W155.13 BOOL  ; EMERG STOP:DEVICE NET COMMUNICATION ABNORMALITY
W155.14 BOOL  ; Servo Carrier Transfer Error
W156.00 BOOL  ; AUTO STOP:INSULATION TESTER FAULT
W156.01 BOOL  ; AUTO STOP:RESISTANCE TESTER FAULT
W156.02 BOOL  ; AUTO STOP:IMPULSE TESTER FAULT
W158.00 BOOL  ; CYCLE STOP:QUALITY CHECK
W159.01 BOOL  ; CYCLE STOP:CONTACT PROBE IN WITHSTAND VOLTAGE FAULT
W159.02 BOOL  ; CYCLE STOP:INSULATION TEST FAULT CONTINUALING
W159.03 BOOL  ; CYCLE STOP:WORK No. FAULT CONTINUALING
W159.04 BOOL  ; CYCLE STOP:SWING MEASUREMENT FAULT CONTINUALING
W159.05 BOOL  ; CYCLE STOP:RESISTANCE MEASUREMENT FAULT CONTINUALING
W159.06 BOOL  ; CYCLE STOP:PAIR POLE IMPULSE MEAS FAULT CONTINUALING
W159.07 BOOL  ; CYCLE STOP:NEXT POLE IMPULSE MEAS FAULT CONTINUALING
W159.08 BOOL  ; CYCLE STOP:LENGTH MEASUREMENT FAULT CONTINUALING
W159.09 BOOL  ; CYCLE STOP:THICKNESS OF CORE FAULT CONTINUALING
W159.10 BOOL  ; CYCLE STOP:COIL END FAULT CONTINUALING
W159.11 BOOL  ; CYCLE STOP:WITHSTAND VOLTAGE CONTACT PROBE CHANGE
W159.12 BOOL  ; CYCLE STOP:RESISTANCE CONTACT PROBE CHANGE
W159.13 BOOL  ; CYCLE STOP:IMPULSE CONTACT PROBE CHANGE
W159.14 BOOL  ; CYCLE STOP:BEARING INSIDE AND OUTSIDE CHECK NG
W159.15 BOOL  ; CYCLE STOP:FULL FRACTION TRAY
W160.00 BOOL  ; CYCLE STOP:LOADING WORKPIECE CLAMP FAULT
W160.01 BOOL  ; CYCLE STOP:UNLOADING WORKPIECE CLAMP FAULT
W160.02 BOOL  ; CYCLE STOP:BEARING MEASUREMENT FAULT CONTINUALING
W160.03 BOOL  ; -
W161.00 BOOL  ; CYCLE STOP:NO WORK No. SWITCH NEXT PRODUCT WORK No.
W163.01 BOOL  ; FAULT STOP:LOADING C/V CYCLE TIME OVER
W163.02 BOOL  ; FAULT STOP:LOADER CYCLE TIME OVER
W163.03 BOOL  ; FAULT STOP:TRANSFER CARRIER CYCLE TIME OVER
W163.04 BOOL  ; FAULT STOP:FWORKPIECE PUSHER CYCLE TIME OVER
W163.05 BOOL  ; FAULT STOP:INSULATION TEST CYCLE TIME OVER
W163.06 BOOL  ; FAULT STOP:SWING MEASUREMENT CYCLE TIME OVER
W163.07 BOOL  ; FAULT STOP:RESISTANCE CYCLE TIME OVER
W163.08 BOOL  ; FAULT STOP:IMPULSE CYCLE TIME OVER
W163.09 BOOL  ; FAULT STOP:BEARING INSERT CYCLE TIME OVER
W163.10 BOOL  ; FAULT STOP:LENGTH MEASUREMENT CYCLE TIME OVER
W163.11 BOOL  ; FAULT STOP:UNLOADING CYCLE TIME OVER
W163.12 BOOL  ; FAULT STOP:BEARING SUPPLY CYCLE TIME OVER
W163.13 BOOL  ; FAULT STOP:BEARING EXCHANGE CYCLE TIME OVER
W163.14 BOOL  ; FAULT STOP:DEFECT DISCHARGE CYCLE TIME OVER
W163.15 BOOL  ; FAULT STOP:LANE 1 PALLETIZING CYCLE TIME OVER
W164.00 BOOL  ; FAULT STOP:LANE 1 SUPPLYING CYCLE TIME OVER
W164.01 BOOL  ; FAULT STOP:LANE 1 STACKING CYCLE TIME OVER
W164.02 BOOL  ; FAULT STOP:LANE 2 PALLETIZING CYCLE TIME OVER
W164.03 BOOL  ; FAULT STOP:LANE 2 SUPPLYING CYCLE TIME OVER
W164.04 BOOL  ; FAULT STOP:LANE 2 STACKING CYCLE TIME OVER
W164.07 BOOL  ; -
W164.08 BOOL  ; -
W166.00 BOOL  ; PAUSE:FULL WORKPIECES OF DEFECT DISCHARGING C/V
W166.01 BOOL  ; PAUSE:LANE 1 FULL UNLOADING CONTAINER
W166.02 BOOL  ; PAUSE:LANE 2 FULL UNLOADING CONTAINER
W166.04 BOOL  ; PAUSE:LANE 1 FULL BEARING TRAY
W166.05 BOOL  ; PAUSE:LANE 1 SHORTAGE OF LOADING CONTAINER
W166.06 BOOL  ; PAUSE:LANE 2 SHORTAGE OF LOADING CONTAINER
W166.08 BOOL  ; PAUSE:SHORTAGE OF BEARING TRAY
W167.00 BOOL  ; NOTICE OF STOP:QUALITY CHECK
W167.01 BOOL  ; NOTICE OF STOP:WITHSTAND VOLTAGE CONTACT PROBE CHANGE
W167.02 BOOL  ; NOTICE OF STOP:RESISTANCE CONTACT PROBE CHANGE
W167.03 BOOL  ; NOTICE OF STOP:IMPULSE CONTACT PROBE CHANGE
W168.00 BOOL  ; PAUSE:WAITING FOR LOADING WORKPIECE
W169.00 BOOL  ; WARNING:SAFETY GUARD OPEN
W169.01 BOOL  ; WARNING:ID COLLATION FAULT OF LOADING CONTAINER
W169.02 BOOL  ; WARNING:SWITCH NEXT WORK No. UNSETTING
W169.03 BOOL  ; WARNING:NO RESPONSE OF ID1
W169.04 BOOL  ; WARNING:COMMUNICATION FAULT OF ID 1
W169.05 BOOL  ; WARNING:NO RESPONSE OF ID2
W169.06 BOOL  ; WARNING:COMMUNICATION FAULT OF ID 2
W169.07 BOOL  ; WARNING:NO RESPONSE OF ID3
W169.08 BOOL  ; WARNING:COMMUNICATION FAULT OF ID 3
W169.09 BOOL  ; WARNING:NO RESPONSE OF ID4
W169.10 BOOL  ; WARNING:COMMUNICATION FAULT OF ID 4
W169.13 BOOL  ; WARNING:BEARING ROBOT BAATERY CHANGE
W169.14 BOOL  ; WARNING:UNLOADING ROBOT BAATERY CHANGE
W169.15 BOOL  ; WARNING:PC BAATERY CHANGE
W170.00 BOOL  ; Defective history clearness
W171.00 BOOL  ; DATA CLEAR
W172.00 BOOL  ; DATA CLEAR
W173.00 BOOL  ; Fraction palette data clearness
W173.11 BOOL  ; Counter effective PB of time
W173.12 BOOL  ; Counter invalid PB of time
W173.13 BOOL  ; Data reset
W173.14 BOOL  ; Stop at one o'clock of utilization rates meter
W174.00 BOOL  ; WORKPIECE MEMORY CLEAR (CORE DISTINCTION UNIT)
W174.01 BOOL  ; WORKPIECE MEMORY CLEAR (INSULATION UNIT)
W174.02 BOOL  ; WORKPIECE MEMORY CLEAR (SWING MEASUREMENT UNIT)
W174.03 BOOL  ; WORKPIECE MEMORY CLEAR (RESISTANCE MEASUREMENT UNIT)
W174.04 BOOL  ; WORKPIECE MEMORY CLEAR (IMPULSE MEASUREMENT UNIT)
W174.05 BOOL  ; WORKPIECE MEMORY CLEAR (BEARING INSERT UNIT)
W174.06 BOOL  ; WORKPIECE MEMORY CLEAR (LENGTH MEASUREMENT UNIT)
W174.07 BOOL  ; WORKPIECE MEMORY CLEAR (UNLOADING UNIT)
W174.08 BOOL  ; WORKPIECE MEMORY CLEAR (ROBOT CHUCK)
W175.10 BOOL  ; Stop at one o'clock of utilization rates meter
W175.11 BOOL  ; Counter effective inside of time
W175.12 BOOL  ; Counter invalid inside of time
W175.14 BOOL  ; It is stopping at one o'clock of the utilization rates meter.
W176.00 BOOL  ; SHORT STOP DATA CLEAR
W176.01 BOOL  ; NO STOP TIME CLEAR
W176.02 BOOL  ; ARMATURE LINE RUNNING
W176.03 BOOL  ; NO STOP TIME COUNT
W176.05 BOOL  ; -
W176.06 BOOL  ; -
W176.07 BOOL  ; -
W176.08 BOOL  ; -
W176.09 BOOL  ; -
W176.10 BOOL  ; -
W18.00 BOOL  ; 11ST_HOME POSITION RETURN PUSH BUTTON SWITCH
W18.01 BOOL  ; 12ST_HOME POSITION RETURN PUSH BUTTON SWITCH
W18.02 BOOL  ; 13ST_HOME POSITION RETURN PUSH BUTTON SWITCH
W18.03 BOOL  ; 14ST_HOME POSITION RETURN PUSH BUTTON SWITCH
W18.04 BOOL  ; 15ST_HOME POSITION RETURN PUSH BUTTON SWITCH
W18.05 BOOL  ; 16ST_HOME POSITION RETURN PUSH BUTTON SWITCH
W18.06 BOOL  ; 17ST_HOME POSITION RETURN PUSH BUTTON SWITCH
W18.07 BOOL  ; 18ST_HOME POSITION RETURN PUSH BUTTON SWITCH
W18.08 BOOL  ; 19ST_HOME POSITION RETURN PUSH BUTTON SWITCH
W18.09 BOOL  ; 20ST_HOME POSITION RETURN PUSH BUTTON SWITCH
W190.00 BOOL  ; ALARM (1ST) PL
W190.01 BOOL  ; ALARM (2ST) PL
W190.02 BOOL  ; ALARM (3ST) PL
W190.03 BOOL  ; ALARM (4ST) PL
W190.04 BOOL  ; ALARM (5ST) PL
W190.05 BOOL  ; ALARM (6ST) PL
W190.06 BOOL  ; ALARM (7ST) PL
W190.07 BOOL  ; ALARM (8ST) PL
W190.08 BOOL  ; ALARM (9ST) PL
W190.09 BOOL  ; ALARM (10ST) PL
W190.10 BOOL  ; ALARM (11ST) PL
W190.11 BOOL  ; ALARM (12ST) PL
W190.12 BOOL  ; ALARM (13ST) PL
W190.13 BOOL  ; ALARM (14ST) PL
W190.14 BOOL  ; ALARM (15ST) PL
W190.15 BOOL  ; ALARM (16ST) PL
W191.00 BOOL  ; CAUTION (1ST) PL
W191.01 BOOL  ; CAUTION (2ST) PL
W191.02 BOOL  ; CAUTION (3ST) PL
W191.03 BOOL  ; CAUTION (4ST) PL
W191.04 BOOL  ; CAUTION (5ST) PL
W191.05 BOOL  ; CAUTION (6ST) PL
W191.06 BOOL  ; CAUTION (7ST) PL
W191.07 BOOL  ; CAUTION (8ST) PL
W191.08 BOOL  ; CAUTION (9ST) PL
W191.09 BOOL  ; CAUTION (10ST) PL
W191.10 BOOL  ; CAUTION (11ST) PL
W191.11 BOOL  ; CAUTION (12ST) PL
W191.12 BOOL  ; CAUTION (13ST) PL
W191.13 BOOL  ; CAUTION (14ST) PL
W191.14 BOOL  ; CAUTION (15ST) PL
W191.15 BOOL  ; CAUTION (16ST) PL
W192.00 BOOL  ; NO FAULT (1ST) PL
W192.01 BOOL  ; NO FAULT (2ST) PL
W192.02 BOOL  ; NO FAULT (3ST) PL
W192.03 BOOL  ; NO FAULT (4ST) PL
W192.04 BOOL  ; NO FAULT (5ST) PL
W192.05 BOOL  ; NO FAULT (6ST) PL
W192.06 BOOL  ; NO FAULT (7ST) PL
W192.07 BOOL  ; NO FAULT (8ST) PL
W192.08 BOOL  ; NO FAULT (9ST) PL
W192.09 BOOL  ; NO FAULT (10ST) PL
W192.10 BOOL  ; NO FAULT (11ST) PL
W192.11 BOOL  ; NO FAULT (12ST) PL
W192.12 BOOL  ; NO FAULT (13ST) PL
W192.13 BOOL  ; NO FAULT (14ST) PL
W192.14 BOOL  ; NO FAULT (15ST) PL
W192.15 BOOL  ; NO FAULT (16ST) PL
W193.00 BOOL  ; ALARM (17ST) PL
W193.01 BOOL  ; ALARM (18ST) PL
W193.02 BOOL  ; ALARM (19ST) PL
W193.03 BOOL  ; ALARM (20ST) PL
W194.00 BOOL  ; CAUTION (17ST) PL
W194.01 BOOL  ; CAUTION (18ST) PL
W194.02 BOOL  ; CAUTION (19ST) PL
W194.03 BOOL  ; CAUTION (20ST) PL
W195.00 BOOL  ; NO FAULT (17ST) PL
W195.01 BOOL  ; NO FAULT (18ST) PL
W195.02 BOOL  ; NO FAULT (19ST) PL
W195.03 BOOL  ; NO FAULT (20ST) PL
W199.08 BOOL  ; SHORT STOP HISTORY SAVE
W199.09 BOOL  ; SHORT STOP HISTORY SAVING
W199.10 BOOL  ; SHORT STOP HISTORY SAVE COMPLETE
W199.11 BOOL  ; SHORT STOP HISTORY SAVE PERMIT
W199.12 BOOL  ; FAULT STOP HISTORY SAVE
W199.13 BOOL  ; FAULT STOP HISTORY SAVING
W199.14 BOOL  ; FAULT STOP HISTORY SAVE COMPLETE
W199.15 BOOL  ; FAULT STOP HISTORY SAVE PERMIT
W19.00 BOOL  ; 11ST_HOME POSITION/RUNNING
W19.01 BOOL  ; 12ST_HOME POSITION/RUNNING
W19.02 BOOL  ; 13ST_HOME POSITION/RUNNING
W19.03 BOOL  ; 14ST_HOME POSITION/RUNNING
W19.04 BOOL  ; 15ST_HOME POSITION/RUNNING
W19.05 BOOL  ; 16ST_HOME POSITION/RUNNING
W19.06 BOOL  ; 17ST_HOME POSITION/RUNNING
W19.07 BOOL  ; 18ST_HOME POSITION/RUNNING
W19.08 BOOL  ; 19ST_HOME POSITION/RUNNING
W19.09 BOOL  ; 20ST_HOME POSITION/RUNNING
W1.00 BOOL  ; MASTER SWITCH ON
W1.01 BOOL  ; AUTO RUNNING
W1.02 BOOL  ; CYCLE STOP
W1.03 BOOL  ; ALL HOME POSITION
W1.04 BOOL  ; OPERATION AUTOMATIC SELECT
W1.05 BOOL  ; OPERATION INDIVIDUAL SELECT
W1.06 BOOL  ; ROBOT 1 RUNNING
W1.07 BOOL  ; ROBOT 2 RUNNING
W1.08 BOOL  ; LS203115
W1.09 BOOL  ; Safety cover invalidity PL
W20.00 BOOL  ; 01ST_HOME POSITION RETURN PUSH BUTTON SWITCH
W20.01 BOOL  ; 02ST_HOME POSITION RETURN PUSH BUTTON SWITCH
W20.02 BOOL  ; 03ST_HOME POSITION RETURN PUSH BUTTON SWITCH
W20.03 BOOL  ; 04ST_HOME POSITION RETURN PUSH BUTTON SWITCH
W20.04 BOOL  ; 05ST_HOME POSITION RETURN PUSH BUTTON SWITCH
W20.05 BOOL  ; 06ST_HOME POSITION RETURN PUSH BUTTON SWITCH
W20.06 BOOL  ; 07ST_HOME POSITION RETURN PUSH BUTTON SWITCH
W20.07 BOOL  ; 08ST_HOME POSITION RETURN PUSH BUTTON SWITCH
W20.08 BOOL  ; 09ST_HOME POSITION RETURN PUSH BUTTON SWITCH
W20.09 BOOL  ; 10ST_HOME POSITION RETURN PUSH BUTTON SWITCH
W21.00 BOOL  ; 01ST_HOME POSITION/RUNNING
W21.01 BOOL  ; 02ST_HOME POSITION/RUNNING
W21.02 BOOL  ; 03ST_HOME POSITION/RUNNING
W21.03 BOOL  ; 04ST_HOME POSITION/RUNNING
W21.04 BOOL  ; 05ST_HOME POSITION/RUNNING
W21.05 BOOL  ; 06ST_HOME POSITION/RUNNING
W21.06 BOOL  ; 07ST_HOME POSITION/RUNNING
W21.07 BOOL  ; 08ST_HOME POSITION/RUNNING
W21.08 BOOL  ; 09ST_HOME POSITION/RUNNING
W21.09 BOOL  ; 10ST_HOME POSITION/RUNNING
W25.00 BOOL  ; LOADING CONVEYOR PALLET SHIFT FORWARD
W25.01 BOOL  ; LOADING CONVEYOR PALLET SHIFT BACKWARD
W25.04 BOOL  ; LOADING CONVEYOR PALLET DISCHARGE FORWARD
W25.05 BOOL  ; LOADING CONVEYOR PALLET DISCHARGE BACKWARD
W26.00 BOOL  ; LOADING CONVEYOR PALLET SHIFT FORWARD END
W26.01 BOOL  ; LOADING CONVEYOR PALLET SHIFT BACKWARD END
W26.04 BOOL  ; LOADING CONVEYOR PALLET DISCHARGE FORWARD END
W26.05 BOOL  ; LOADING CONVEYOR PALLET DISCHARGE BACKWARD END
W27.00 BOOL  ; WORKPIECE ON FORMER PROCESS
W27.10 BOOL  ; 01ST_1CY START PB
W27.11 BOOL  ; 01ST_1CY RUN PL
W27.12 BOOL  ; 01ST_UNIT HOME POSITION RETURN PB
W27.13 BOOL  ; 01ST_UNIT HOME POSITION PL
W28.00 BOOL  ; LOADER FORWARD
W28.01 BOOL  ; LOADER BACKWARD
W28.02 BOOL  ; LOADER DOWNWARD
W28.03 BOOL  ; LOADER UPWARD
W28.04 BOOL  ; TURN LOADER CHUCK TURN
W28.05 BOOL  ; TURN LOADER RECHUCK TURN
W28.06 BOOL  ; LOADER CHUCK CLAMP
W28.07 BOOL  ; LOADER CHUCK UNCLAMP
W29.00 BOOL  ; LOADER FORWARD END
W29.01 BOOL  ; LOADER BACKWARD END
W29.02 BOOL  ; LOADER DOWNWARD END
W29.03 BOOL  ; LOADER UPWARD END
W29.04 BOOL  ; TURN LOADER CHUCK TURN END
W29.05 BOOL  ; TURN LOADER CHUCK RETURN END
W29.06 BOOL  ; LOADER CHUCK CLAMP END
W29.07 BOOL  ; LOADER CHUCK UNCLAMP END
W2.01 BOOL  ; $?St$Bk?_#[22] / PB_Upper limit master check / $?St$Bk?_#[22]
W2.02 BOOL  ; ROBOT MASTER ON
W2.03 BOOL  ; ROBOT FIXED POSITION RETURN
W2.04 BOOL  ; LENGTH MASTER O SETTING
W2.05 BOOL  ; BEARING FIXID POSITION RETURN
W2.06 BOOL  ; ALL MACHINES SAVING ENERGY OF FLURESCENT LIGHT
W2.07 BOOL  ; PB_Lower limit master check
W2.09 BOOL  ; LANGUAGE CHANGE PB
W2.10 BOOL  ; SAVING ENERGY OF FLURESCENT LIGHT
W300.00 BOOL  ; Piling up one lane step lot end(four steps)
W300.01 BOOL  ; Piling up two lane step lot end(four steps)
W300.02 BOOL  ; ID RESET START SELECT PB ON
W300.03 BOOL  ; ID RESET START
W300.04 BOOL  ; ID RESET RUNNING
W301.00 BOOL  ; TEMPORARY CONTACT FOR ADJUSTMENT ON
W301.01 BOOL  ; Product number change 1 （for disp）
W301.02 BOOL  ; Crear product number change 1 （for disp）
W301.05 BOOL  ; -
W301.06 BOOL  ; -
W301.10 BOOL  ; -
W301.15 BOOL  ; 調整用仮接点（ﾜｰｸ押さえ上昇ﾀｲﾐﾝｸﾞ）
W302.01 BOOL  ; Product number change 2 （for disp）
W302.02 BOOL  ; Crear product number change 2 （for disp）
W302.10 BOOL  ; -
W30.00 BOOL  ; TRANSFER CARRIER NO INTERFERENCE
W30.10 BOOL  ; 02ST_1CY START PB
W30.11 BOOL  ; 02ST_1CY RUN PL
W30.12 BOOL  ; 02ST_UNIT HOME POSITION RETURN PB
W30.13 BOOL  ; 02ST_UNIT HOME POSITION PL
W31.00 BOOL  ; TRANSFER CARRIER LIFT UPWARD
W31.01 BOOL  ; TRANSFER CARRIER LIFT DOWNWARD
W31.02 BOOL  ; TRANSFER CARRIER FORWARD
W31.03 BOOL  ; TRANSFER CARRIER BACKWARD
W32.00 BOOL  ; TRANSFER CARRIER LIFT UPWARD END
W32.01 BOOL  ; TRANSFER CARRIER LIFT DOWNWARD END
W32.02 BOOL  ; TRANSFER CARRIER FORWARD END
W32.03 BOOL  ; TRANSFER CARRIER BACKWARD END
W33.00 BOOL  ; Completion of distinction of thickness in core
W33.01 BOOL  ; INSULATION TEST COMPLETE
W33.02 BOOL  ; SWING & COIL END COMPLETE
W33.03 BOOL  ; RESISTANCE MEASUREMENT COMPLETE
W33.04 BOOL  ; IMPULSE COMPLETE
W33.05 BOOL  ; BEARING INSERT COMPLETE
W33.06 BOOL  ; LENGTH CHECK COMPLETE
W33.10 BOOL  ; 03ST_1CY START PB
W33.11 BOOL  ; 03ST_1CY RUN PL
W33.12 BOOL  ; 03ST_UNIT HOME POSITION RETURN PB
W33.13 BOOL  ; 03ST_UNIT HOME POSITION PL
W34.00 BOOL  ; WORKPIECE PUSHER FORWARD
W34.01 BOOL  ; WORKPIECE PUSHER BACKWARD
W34.04 BOOL  ; Start of distinction of thickness in core
W34.05 BOOL  ; Stop of distinction of thickness in core
W350.00 BOOL  ; -
W351.00 BOOL  ; -
W35.00 BOOL  ; WORKPIECE PUSHER FORWARD
W35.01 BOOL  ; WORKPIECE PUSHER BACKWARD
W35.04 BOOL  ; Start of distinction of thickness in core
W35.05 BOOL  ; Stop of distinction of thickness in core
W36.01 BOOL  ; Completion of distinction of thickness in core
W36.10 BOOL  ; 04ST_1CY START PB
W36.11 BOOL  ; 04ST_1CY RUN PL
W36.12 BOOL  ; 04ST_UNIT HOME POSITION RETURN PB
W36.13 BOOL  ; 04ST_UNIT HOME POSITION PL
W37.00 BOOL  ; TRANSFER CARRIER LIFT UPWARD
W37.01 BOOL  ; TRANSFER CARRIER LIFT DOWNWARD
W37.04 BOOL  ; INSULATION TEST START
W37.05 BOOL  ; INSULATION TEST STOP
W38.00 BOOL  ; TRANSFER CARRIER LIFT UPWARD END
W38.01 BOOL  ; TRANSFER CARRIER LIFT DOWNWARD END
W38.04 BOOL  ; INSULATION TEST START
W38.05 BOOL  ; INSULATION TEST STOP
W39.01 BOOL  ; INSULATION TEST OK
W39.02 BOOL  ; INSULATION TEST NG
W39.03 BOOL  ; INSULATION TEST COMPLETE
W39.10 BOOL  ; 05ST_1CY START PB
W39.11 BOOL  ; 05ST_1CY RUN PL
W39.12 BOOL  ; 05ST_UNIT HOME POSITION RETURN PB
W39.13 BOOL  ; 05ST_UNIT HOME POSITION PL
W3.01 BOOL  ; PL_Upper limit check completed (functional check)
W3.02 BOOL  ; ROBOT MASTER ON
W3.03 BOOL  ; ROBOT FIXED POSITION PL
W3.04 BOOL  ; PL_LENGTH 0 MASTER SETTING
W3.05 BOOL  ; BEARING FIXID POSITION PL
W3.06 BOOL  ; ALL MACHINES SAVING ENERGY OF FLURESCENT LIGHT
W3.07 BOOL  ; PL_Lower limit check completed (functional check)
W3.10 BOOL  ; SAVING ENERGY OF FLURESCENT LIGHT
W3.11 BOOL  ; SAVING ENERGY OF FLURESCENT LIGHT
W400.00 BOOL  ; TRANSFER +JOG
W400.01 BOOL  ; TRANSFER -JOG
W400.03 BOOL  ; FORWARD POSITION S
W400.04 BOOL  ; BACKWARD POSITION S
W400.07 BOOL  ; Set Up
W400.15 BOOL  ; POSITIONAL DATA CAN BE INPUT
W40.00 BOOL  ; TRANSFER CARRIER LIFT UPWARD
W40.01 BOOL  ; TRANSFER CARRIER LIFT DOWNWARD
W40.02 BOOL  ; POSITIONING ARROW FORWARD
W40.03 BOOL  ; POSITIONING ARROW BACKWARD
W40.04 BOOL  ; POSITIONING START
W40.05 BOOL  ; POSITIONING STOP
W40.08 BOOL  ; SWING MEASURE START
W40.09 BOOL  ; SWING MEASURE STOP
W41.00 BOOL  ; TRANSFER CARRIER LIFT UPWARD END
W41.01 BOOL  ; TRANSFER CARRIER LIFT DOWNWARDD END
W41.02 BOOL  ; POSITIONING ARROW FORWARDD END
W41.03 BOOL  ; POSITIONING ARROW BACKWARDD END
W41.04 BOOL  ; POSITIONING START
W41.05 BOOL  ; POSITIONING STOP
W41.08 BOOL  ; SWING MEASURE START
W41.09 BOOL  ; SWING MEASURE STOP
W42.01 BOOL  ; SWING OK
W42.02 BOOL  ; SWING NG
W42.03 BOOL  ; SWING & COIL END COMPLETE
W42.10 BOOL  ; 06ST_1CY START PB
W42.11 BOOL  ; 06ST_1CY RUN PL
W42.12 BOOL  ; 06ST_UNIT HOME POSITION RETURN PB
W42.13 BOOL  ; 06ST_UNIT HOME POSITION PL
W43.02 BOOL  ; WORKPIECE CLAMP DOWNWARD
W43.03 BOOL  ; WORKPIECE CLAMP UPWARD
W43.06 BOOL  ; TRANSFER CARRIER LIFT UPWARD
W43.07 BOOL  ; TRANSFER CARRIER LIFT DOWNWARD
W43.10 BOOL  ; CONTACT PROBE IN RESISTANCE FORWARD
W43.11 BOOL  ; CONTACT PROBE IN RESISTANCE BACKWARD
W43.14 BOOL  ; RESISTANCE MEASUREMENT START
W43.15 BOOL  ; RESISTANCE MEASUREMENT STOP
W44.02 BOOL  ; TRANSFER CARRIER LIFT UPWARD END
W44.03 BOOL  ; TRANSFER CARRIER LIFT DOWNWARD END
W44.06 BOOL  ; CONTACT PROBE IN RESISTANCE FORWARD END
W44.07 BOOL  ; CONTACT PROBE IN RESISTANCE BACKWARD END
W44.10 BOOL  ; CONTACT PROBE IN RESISTANCE FORWARD END
W44.11 BOOL  ; CONTACT PROBE IN RESISTANCE BACKWARD END
W44.14 BOOL  ; RESISTANCE MEASUREMENT START
W44.15 BOOL  ; RESISTANCE MEASUREMENT STOP
W45.01 BOOL  ; RESISTANCE OK (80)
W45.02 BOOL  ; RESISTANCE NG (80)
W45.03 BOOL  ; RESISTANCE OK (180)
W45.04 BOOL  ; RESISTANCE NG (180)
W45.05 BOOL  ; RESISTANCE MEASUREMENT COMPLETE
W45.10 BOOL  ; 07ST_1CY START PB
W45.11 BOOL  ; 07ST_1CY RUN PL
W45.12 BOOL  ; 07ST_UNIT HOME POSITION RETURN PB
W45.13 BOOL  ; 07ST_UNIT HOME POSITION PL
W46.00 BOOL  ; WORKPIECE CLAMP DOWNWARD
W46.01 BOOL  ; WORKPIECE CLAMP UPWARD
W46.02 BOOL  ; CONTACT PROBE IN INPULSE FORWARD
W46.03 BOOL  ; CONTACT PROBE IN INPULSE BACKWARD
W46.04 BOOL  ; TRANSFER CARRIER LIFT UPWARD
W46.05 BOOL  ; TRANSFER CARRIER LIFT DOWNWARD
W46.06 BOOL  ; IMPULSE MEASUREMENT START
W46.07 BOOL  ; IMPULSE MEASUREMENT STOP
W46.09 BOOL  ; WABE INDICATION
W46.10 BOOL  ; Relay ON to pair pole
W46.11 BOOL  ; Relay ON to next pole
W46.14 BOOL  ; STEP MODE ON
W46.15 BOOL  ; STEP UP
W47.00 BOOL  ; WORKPIECE CLAMP DOWNWARD END
W47.01 BOOL  ; WORKPIECE CLAMP UPWARD END
W47.02 BOOL  ; CONTACT PROBE IN INPULSE FORWARD END
W47.03 BOOL  ; CONTACT PROBE IN INPULSE BACKWARD END
W47.04 BOOL  ; TRANSFER CARRIER LIFT UPWARD END
W47.05 BOOL  ; TRANSFER CARRIER LIFT DOWNWARD END
W47.06 BOOL  ; IMPULSE MEASUREMENT START
W47.07 BOOL  ; IMPULSE MEASUREMENT STOP
W47.09 BOOL  ; WABE INDICATION
W47.10 BOOL  ; Relay ON to pair pole
W47.11 BOOL  ; Relay ON to next pole
W47.14 BOOL  ; STEP MODE ON
W47.15 BOOL  ; STEP UP
W48.01 BOOL  ; PAIR POLE OK
W48.02 BOOL  ; PAIR POLE NG
W48.03 BOOL  ; NEXT POLE OK
W48.04 BOOL  ; NEXT POLE NG
W48.05 BOOL  ; IMPULSE COMPLETE
W48.10 BOOL  ; 08ST_1CY START PB
W48.11 BOOL  ; 08ST_1CY RUN PL
W48.12 BOOL  ; 08ST_UNIT HOME POSITION RETURN PB
W48.13 BOOL  ; 08ST_UNIT HOME POSITION PL
W49.00 BOOL  ; SUB TRANSFER CARRIER LIFT UPWARD
W49.01 BOOL  ; SUB TRANSFER CARRIER LIFT DOWNWARD
W49.02 BOOL  ; BEARING INSERT (HIGH SPEED) FORWARD
W49.03 BOOL  ; BEARING INSERT (HIGH SPEED) BACKWARD
W49.04 BOOL  ; BEARING INSERT (HIGH PRESSURE) ON
W49.05 BOOL  ; BEARING INSERT (HIGH PRESSURE) OFF
W49.06 BOOL  ; BEARING SHUTTER DOWNWARD
W49.07 BOOL  ; BEARING SHUTTER UPWARD
W49.08 BOOL  ; BEARING GUIDE FORWARD
W49.09 BOOL  ; BEARING GUIDE BACKWARD
W49.10 BOOL  ; BEARING ESCAPE FORWARD
W49.11 BOOL  ; BEARING ESCAPE BACKWARD
W49.12 BOOL  ; PB_Work Clamp Downword
W49.13 BOOL  ; PB_Work Clamp Upword
W4.01 BOOL  ; ROBOT FIXED POSITION PL
W4.02 BOOL  ; ROBOT READY
W4.03 BOOL  ; BEARING FIXID POSITION PL
W50.00 BOOL  ; SUB TRANSFER CARRIER LIFT UPWARD
W50.01 BOOL  ; SUB TRANSFER CARRIER LIFT DOWNWARD
W50.02 BOOL  ; BEARING INSERT (HIGH SPEED) FORWARD
W50.03 BOOL  ; BEARING INSERT (HIGH SPEED) BACKWARD
W50.04 BOOL  ; BEARING INSERT (HIGH PRESSURE) ON
W50.05 BOOL  ; BEARING INSERT (HIGH PRESSURE) OFF
W50.06 BOOL  ; BEARING SHUTTER DOWNWARD
W50.07 BOOL  ; BEARING SHUTTER UPWARD
W50.08 BOOL  ; BEARING GUIDE FORWARD
W50.09 BOOL  ; BEARING GUIDE BACKWARD
W50.10 BOOL  ; BEARING ESCAPE FORWARD
W50.11 BOOL  ; BEARING ESCAPE BACKWARD
W50.12 BOOL  ; Work Clamp Downword
W50.13 BOOL  ; Work Clamp Upword
W51.01 BOOL  ; BEARING INSERT COMPLETE
W51.10 BOOL  ; 09ST_1CY START PB
W51.11 BOOL  ; 09ST_1CY RUN PL
W51.12 BOOL  ; 09ST_UNIT HOME POSITION RETURN PB
W51.13 BOOL  ; 09ST_UNIT HOME POSITION PL
W52.00 BOOL  ; SUB TRANSFER CARRIER LIFT UPWARD
W52.01 BOOL  ; SUB TRANSFER CARRIER LIFT DOWNWARD
W52.02 BOOL  ; Work Clamp DownWard
W52.03 BOOL  ; Work Clamp UpWard
W52.04 BOOL  ; LENGTH MEASUREMENT FORWARD
W52.05 BOOL  ; LENGTH MEASUREMENT BACKWARD
W52.08 BOOL  ; LENGTH CHECK START
W52.09 BOOL  ; LENGTH CHECK STOP
W53.00 BOOL  ; SUB TRANSFER CARRIER LIFT UPWARD END
W53.01 BOOL  ; SUB TRANSFER CARRIER LIFT DOWNWARD END
W53.02 BOOL  ; Work Clamp Downword
W53.03 BOOL  ; Work Clamp Upword
W53.04 BOOL  ; LENGTH MEASUREMENT FORWARD END
W53.05 BOOL  ; LENGTH MEASUREMENT BACKWARD END
W53.08 BOOL  ; LENGTH CHECK START
W53.09 BOOL  ; LENGTH CHECK STOP
W54.01 BOOL  ; OVERALL LENGTH OK
W54.02 BOOL  ; OVERALL LENGTH NG
W54.03 BOOL  ; BEARING INSERT LENGTH OK
W54.04 BOOL  ; BEARING INSERT LENGTH NG
W54.05 BOOL  ; LENGTH CHECK COMPLETE
W54.10 BOOL  ; 10ST_1CY START PB
W54.11 BOOL  ; 10ST_1CY RUN PL
W54.12 BOOL  ; 10ST_UNIT HOME POSITION RETURN PB
W54.13 BOOL  ; 10ST_UNIT HOME POSITION PL
W55.00 BOOL  ; UNLOADING ROBOT CHUCK CLAMP
W55.01 BOOL  ; UNLOADING ROBOT CHUCK UNCLAMP
W55.04 BOOL  ; Start of the fraction workpiece is discharged
W56.00 BOOL  ; UNLOADING ROBOT CHUCK CLAMP END
W56.01 BOOL  ; UNLOADING ROBOT CHUCK UNCLAMP END
W56.04 BOOL  ; Start of the fraction workpiece is discharged
W57.01 BOOL  ; UNLOADING UNIT HOME POSITION
W57.02 BOOL  ; ROBOT MASTER ON
W57.03 BOOL  ; FRACTION TRAY CONFIRMATION
W57.10 BOOL  ; 11ST_1CY START PB
W57.11 BOOL  ; 11ST_1CY RUN PL
W57.12 BOOL  ; 11ST_UNIT HOME POSITION RETURN PB
W57.13 BOOL  ; 11ST_UNIT HOME POSITION PL
W58.00 BOOL  ; BEARING TRANSFER CARRIER FORWARD
W58.01 BOOL  ; BEARING TRANSFER CARRIER BACKWARD
W58.02 BOOL  ; BEARING SUPPLY ROBOT TAKING OUT POSITION
W58.03 BOOL  ; BEARING SUPPLY ROBOT HOME POSITION
W58.04 BOOL  ; BEARING HANGER FORWARD
W58.05 BOOL  ; BEARING HANGER BACKWARD
W58.06 BOOL  ; BEARING HANGER DOWNWARD
W58.07 BOOL  ; BEARING HANGER UPWARD
W58.08 BOOL  ; BEARING TRANSFER UPWARD
W58.09 BOOL  ; BEARING TRANSFER DOWNWARD
W58.10 BOOL  ; BEARING PUSHER BACKWARD
W58.11 BOOL  ; BEARING PUSHER FORWARD
W59.00 BOOL  ; BEARING TRANSFER CARRIER FORWARD END
W59.01 BOOL  ; BEARING TRANSFER CARRIER BACKWARD END
W59.02 BOOL  ; BEARING SUPPLY ROBOT TAKING OUT POSITION
W59.03 BOOL  ; BEARING SUPPLY ROBOT HOME POSITION
W59.04 BOOL  ; BEARING HANGER FORWARD END
W59.05 BOOL  ; BEARING HANGER BACKWARD END
W59.06 BOOL  ; BEARING HANGER DOWNWARD END
W59.07 BOOL  ; BEARING HANGER UPWARD END
W59.08 BOOL  ; BEARING TRANSFER UPWARD END
W59.09 BOOL  ; BEARING TRANSFER DOWNWARD END
W59.10 BOOL  ; BEARING PUSHER BACKWARD END
W59.11 BOOL  ; BEARING PUSHER FORWARD END
W5.01 BOOL  ; MASTER SWITCH OFF
W5.02 BOOL  ; MASTER SETTING PB
W5.04 BOOL  ; NG WORKPIECE INSULATION TEST PB
W5.05 BOOL  ; NG WORKPIECE IMPULSE MEASURE
W5.06 BOOL  ; NG WORKPIECE SWING MEASURE
W5.07 BOOL  ; NG WORKPIECE BEARING INSERT
W5.08 BOOL  ; NG WORKPIECE RESISTANCE MEASURE
W5.09 BOOL  ; NG WORKPIECE LENGTH MEASURE
W60.01 BOOL  ; BEARING TRAY CONFIRMATION
W60.10 BOOL  ; 12ST_1CY START PB
W60.11 BOOL  ; 12ST_1CY RUN PL
W60.12 BOOL  ; 12ST_UNIT HOME POSITION RETURN PB
W60.13 BOOL  ; 12ST_UNIT HOME POSITION PL
W61.00 BOOL  ; BEARING TRAY HOME POSITIONING BACKWARD
W61.01 BOOL  ; BEARING TRAY HOME POSITIONING FORWARD
W61.02 BOOL  ; BEARING TRAY EXCHANGE DOWNWARD
W61.03 BOOL  ; BEARING TRAY EXCHANGE UPWARD
W61.04 BOOL  ; BEARING TRAY STOPPER BACKWARD
W61.05 BOOL  ; BEARING TRAY STOPPER FORWARD
W61.06 BOOL  ; BEARING TRAY ESCAPE FORWARD
W61.07 BOOL  ; BEARING TRAY ESCAPE BACKWARD
W61.08 BOOL  ; EXCHANGE CONVEYOR CW ROTATE
W61.09 BOOL  ; EXCHANGE CONVEYOR CCW ROTATE
W61.12 BOOL  ; LOADING CONVEYOR ON
W61.13 BOOL  ; UNLOADING CONVEYOR ON
W61.14 BOOL  ; CONVEYOR OFF
W62.00 BOOL  ; BEARING TRAY HOME POSITIONING FORWARD END
W62.01 BOOL  ; BEARING TRAY HOME POSITIONING BACKWARD END
W62.02 BOOL  ; BEARING TRAY EXCHANGE DOWNWARD END
W62.03 BOOL  ; BEARING TRAY EXCHANGE UPWARD END
W62.04 BOOL  ; BEARING TRAY STOPPER BACKWARD END
W62.05 BOOL  ; BEARING TRAY STOPPER FORWARD END
W62.06 BOOL  ; BEARING TRAY ESCAPE FORWARD END
W62.07 BOOL  ; BEARING TRAY ESCAPE BACKWARD END
W62.08 BOOL  ; EXCHANGE CONVEYOR CW ROTATE
W62.09 BOOL  ; EXCHANGE CONVEYOR CCW ROTATE
W62.12 BOOL  ; LOADING CONVEYOR ON
W62.13 BOOL  ; UNLOADING CONVEYOR ON
W62.14 BOOL  ; CONVEYOR OFF
W63.01 BOOL  ; TAKING OUT COMPLETE
W63.05 BOOL  ; NO INTERFERENCE OF BEARING SUPPLY ROBOT
W63.10 BOOL  ; 13ST_1CY START PB
W63.11 BOOL  ; 13ST_1CY RUN PL
W63.12 BOOL  ; 13ST_UNIT HOME POSITION RETURN PB
W63.13 BOOL  ; 13ST_UNIT HOME POSITION PL
W64.00 BOOL  ; DEFECT CONVEYOR ON
W65.00 BOOL  ; DEFECT CONVEYOR OFF
W66.10 BOOL  ; 14ST_1CY START PB
W66.11 BOOL  ; 14ST_1CY RUN PL
W66.12 BOOL  ; 14ST_UNIT HOME POSITION RETURN PB
W66.13 BOOL  ; 14ST_UNIT HOME POSITION PL
W67.00 BOOL  ; CONVEYOR START AFTER PALLETIZING
W67.01 BOOL  ; CONVEYOR STOP AFTER PALLETIZING
W67.02 BOOL  ; STOPPER BEFOR PALLETIZING DOWNWARD
W67.03 BOOL  ; STOPPER BEFOR PALLETIZING UPWARD
W67.04 BOOL  ; PALLETIZING HOOK BACKWARD
W67.05 BOOL  ; PALLETIZING HOOK FORWARD
W67.06 BOOL  ; PALLETIZING LIFTER DOWNWARD
W67.07 BOOL  ; PALLETIZING LIFTER UPWARD
W67.08 BOOL  ; PALLETIZING CONVEYOR
W67.10 BOOL  ; STOPPER BEFOR PALLETIZING DOWNWARD
W67.11 BOOL  ; STOPPER BEFOR PALLETIZING UPWARD
W67.12 BOOL  ; LOADING CONVEYOR
W67.14 BOOL  ; ESCAPE BEFOR PALLETIZING UPWARD
W67.15 BOOL  ; ESCAPE BEFOR PALLETIZING DOWNWARD
W68.00 BOOL  ; CONVEYOR START AFTER PALLETIZING
W68.01 BOOL  ; CONVEYOR STOP AFTER PALLETIZING
W68.02 BOOL  ; STOPPER BEFOR PALLETIZING DOWNWARD END
W68.03 BOOL  ; STOPPER BEFOR PALLETIZING UPWARD END
W68.04 BOOL  ; PALLETIZING HOOK BACKWARD END
W68.05 BOOL  ; PALLETIZING HOOK FORWARD END
W68.06 BOOL  ; PALLETIZING LIFTER DOWNWARD END
W68.07 BOOL  ; PALLETIZING LIFTER UPWARD END
W68.08 BOOL  ; PALLETIZING CONVEYOR
W68.10 BOOL  ; STOPPER BEFOR PALLETIZING DOWNWARD END
W68.11 BOOL  ; STOPPER BEFOR PALLETIZING UPWARD END
W68.12 BOOL  ; LOADING CONVEYOR
W68.14 BOOL  ; ESCAPE BEFOR PALLETIZING UPWARD END
W68.15 BOOL  ; ESCAPE BEFOR PALLETIZING DOWNWARD END
W69.10 BOOL  ; 15ST_1CY START PB
W69.11 BOOL  ; 15ST_1CY RUN PL
W69.12 BOOL  ; 15ST_UNIT HOME POSITION RETURN PB
W69.13 BOOL  ; 15ST_UNIT HOME POSITION PL
W6.02 BOOL  ; MASTER SETTING
W6.04 BOOL  ; NG WORKPIECE INSULATION TEST
W6.05 BOOL  ; NG WORKPIECE IMPULSE MEASURE
W6.06 BOOL  ; NG WORKPIECE SWING MEASURE
W6.07 BOOL  ; NG WORKPIECE BEARING INSERT
W6.08 BOOL  ; NG WORKPIECE RESISTANCE MEASURE
W6.09 BOOL  ; NG WORKPIECE LENGTH MEASURE
W70.00 BOOL  ; POSITIONING 1 BACKWARD
W70.01 BOOL  ; POSITIONING 1 FORWARD
W70.02 BOOL  ; LIFTER DOWNWARD
W70.03 BOOL  ; LIFTER UPWARD
W70.04 BOOL  ; POSITIONING 2 BACKWARD
W70.05 BOOL  ; POSITIONING 2 FORWARD
W70.06 BOOL  ; DROP GUARD BACKWARD
W70.07 BOOL  ; DROP GUARD FORWARD
W70.08 BOOL  ; EXCHANGE CONVEYOR CW
W70.09 BOOL  ; EXCHANGE CONVEYOR CCW
W70.10 BOOL  ; Writing of ID1
W70.11 BOOL  ; Writing of ID2
W70.12 BOOL  ; PALLETIZING CONVEYOR
W70.13 BOOL  ; STACKING CONVEYOR
W70.14 BOOL  ; CONVEYOR STOP
W71.00 BOOL  ; POSITIONING 1 BACKWARD END
W71.01 BOOL  ; POSITIONING 1 FORWARD END
W71.02 BOOL  ; LIFTER DOWNWARD END
W71.03 BOOL  ; LIFTER UPWARD END
W71.04 BOOL  ; POSITIONING 2 BACKWARD END
W71.05 BOOL  ; POSITIONING 2 FORWARD END
W71.06 BOOL  ; DROP GUARD BACKWARD END
W71.07 BOOL  ; DROP GUARD FORWARD END
W71.08 BOOL  ; EXCHANGE CONVEYOR CW
W71.09 BOOL  ; EXCHANGE CONVEYOR CCW
W71.10 BOOL  ; Writing completion of ID1
W71.11 BOOL  ; Writing completion of ID2
W71.12 BOOL  ; PALLETIZING CONVEYOR
W71.13 BOOL  ; STACKING CONVEYOR
W71.14 BOOL  ; CONVEYOR STOP
W72.05 BOOL  ; NO INTERFERENCE OF ROBOT
W72.10 BOOL  ; 16ST_1CY START PB
W72.11 BOOL  ; 16ST_1CY RUN PL
W72.12 BOOL  ; 16ST_UNIT HOME POSITION RETURN PB
W72.13 BOOL  ; 16ST_UNIT HOME POSITION PL
W73.00 BOOL  ; STACKING HOOK BACKWARD
W73.01 BOOL  ; STACKING HOOK FORWARD
W73.02 BOOL  ; STACKING LIFTER DOWNWARD
W73.03 BOOL  ; STACKING LIFTER UPWARD
W73.04 BOOL  ; STACKING CONVEYOR
W73.05 BOOL  ; CONVEYOR STOP
W73.06 BOOL  ; STACKING STOPPER DOWNWARD
W73.07 BOOL  ; STACKING STOPPER UPWARD
W73.08 BOOL  ; UNLOADING CONVEYOR 1
W73.10 BOOL  ; UNLOADING ESCAPE UPWARD
W73.11 BOOL  ; UNLOADING ESCAPE DOWNWARD
W73.12 BOOL  ; UNLOADING CONVEYOR 2
W73.14 BOOL  ; UNLOADING STOPPER DOWNWARD
W73.15 BOOL  ; UNLOADING STOPPER UPWARD
W74.00 BOOL  ; STACKING HOOK BACKWARD END
W74.01 BOOL  ; STACKING HOOK FORWARD END
W74.02 BOOL  ; STACKING LIFTER DOWNWARD END
W74.03 BOOL  ; STACKING LIFTER UPWARD END
W74.04 BOOL  ; STACKING CONVEYOR
W74.05 BOOL  ; CONVEYOR STOP
W74.06 BOOL  ; STACKING STOPPER DOWNWARD END
W74.07 BOOL  ; STACKING STOPPER UPWARD END
W74.08 BOOL  ; UNLOADING CONVEYOR 1
W74.10 BOOL  ; UNLOADING ESCAPE UPWARD END
W74.11 BOOL  ; UNLOADING ESCAPE DOWNWARD END
W74.12 BOOL  ; UNLOADING CONVEYOR 2
W74.14 BOOL  ; UNLOADING STOPPER DOWNWARD END
W74.15 BOOL  ; UNLOADING STOPPER UPWARD END
W75.10 BOOL  ; 17ST_1CY START PB
W75.11 BOOL  ; 17ST_1CY RUN PL
W75.12 BOOL  ; 17ST_UNIT HOME POSITION RETURN PB
W75.13 BOOL  ; 17ST_UNIT HOME POSITION PL
W76.00 BOOL  ; CONVEYOR START AFTER PALLETIZING
W76.01 BOOL  ; CONVEYOR STOP AFTER PALLETIZING
W76.02 BOOL  ; STOPPER BEFOR PALLETIZING DOWNWARD
W76.03 BOOL  ; STOPPER BEFOR PALLETIZING UPWARD
W76.04 BOOL  ; PALLETIZING HOOK BACKWARD
W76.05 BOOL  ; PALLETIZING HOOK FORWARD
W76.06 BOOL  ; PALLETIZING LIFTER DOWNWARD
W76.07 BOOL  ; PALLETIZING LIFTER UPWARD
W76.08 BOOL  ; PALLETIZING CONVEYOR
W76.10 BOOL  ; STOPPER BEFOR PALLETIZING DOWNWARD
W76.11 BOOL  ; STOPPER BEFOR PALLETIZING UPWARD
W76.12 BOOL  ; LOADING CONVEYOR
W76.14 BOOL  ; ESCAPE BEFOR PALLETIZING UPWARD
W76.15 BOOL  ; ESCAPE BEFOR PALLETIZING DOWNWARD
W77.00 BOOL  ; CONVEYOR START AFTER PALLETIZING
W77.01 BOOL  ; CONVEYOR STOP AFTER PALLETIZING
W77.02 BOOL  ; STOPPER BEFOR PALLETIZING DOWNWARD END
W77.03 BOOL  ; STOPPER BEFOR PALLETIZING UPWARD END
W77.04 BOOL  ; PALLETIZING HOOK BACKWARD END
W77.05 BOOL  ; PALLETIZING HOOK FORWARD END
W77.06 BOOL  ; PALLETIZING LIFTER DOWNWARD END
W77.07 BOOL  ; PALLETIZING LIFTER UPWARD END
W77.08 BOOL  ; PALLETIZING CONVEYOR
W77.10 BOOL  ; STOPPER BEFOR PALLETIZING DOWNWARD END
W77.11 BOOL  ; STOPPER BEFOR PALLETIZING UPWARD END
W77.12 BOOL  ; LOADING CONVEYOR
W77.14 BOOL  ; ESCAPE BEFOR PALLETIZING UPWARD END
W77.15 BOOL  ; ESCAPE BEFOR PALLETIZING DOWNWARD END
W78.10 BOOL  ; 18ST_1CY START PB
W78.11 BOOL  ; 18ST_1CY RUN PL
W78.12 BOOL  ; 18ST_UNIT HOME POSITION RETURN PB
W78.13 BOOL  ; 18ST_UNIT HOME POSITION PL
W79.00 BOOL  ; POSITIONING 1 BACKWARD
W79.01 BOOL  ; POSITIONING 1 FORWARD
W79.02 BOOL  ; LIFTER DOWNWARD
W79.03 BOOL  ; LIFTER UPWARD
W79.04 BOOL  ; POSITIONING 2 BACKWARD
W79.05 BOOL  ; POSITIONING 2 FORWARD
W79.06 BOOL  ; DROP GUARD BACKWARD
W79.07 BOOL  ; DROP GUARD FORWARD
W79.08 BOOL  ; EXCHANGE CONVEYOR CW
W79.09 BOOL  ; EXCHANGE CONVEYOR CCW
W79.10 BOOL  ; Writing of ID3
W79.11 BOOL  ; Writing of ID4
W79.12 BOOL  ; PALLETIZING CONVEYOR
W79.13 BOOL  ; STACKING CONVEYOR
W79.14 BOOL  ; CONVEYOR STOP
W80.00 BOOL  ; POSITIONING 1 BACKWARD END
W80.01 BOOL  ; POSITIONING 1 FORWARD END
W80.02 BOOL  ; LIFTER DOWNWARD END
W80.03 BOOL  ; LIFTER UPWARD END
W80.04 BOOL  ; POSITIONING 2 BACKWARD END
W80.05 BOOL  ; POSITIONING 2 FORWARD END
W80.06 BOOL  ; DROP GUARD BACKWARD END
W80.07 BOOL  ; DROP GUARD FORWARD END
W80.08 BOOL  ; EXCHANGE CONVEYOR CW
W80.09 BOOL  ; EXCHANGE CONVEYOR CCW
W80.10 BOOL  ; Writing completion of ID3
W80.11 BOOL  ; Writing completion of ID4
W80.12 BOOL  ; PALLETIZING CONVEYOR
W80.13 BOOL  ; STACKING CONVEYOR
W80.14 BOOL  ; CONVEYOR STOP
W81.05 BOOL  ; NO INTERFERENCE OF ROBOT
W81.10 BOOL  ; 19ST_1CY START PB
W81.11 BOOL  ; 19ST_1CY RUN PL
W81.12 BOOL  ; 19ST_UNIT HOME POSITION RETURN PB
W81.13 BOOL  ; 19ST_UNIT HOME POSITION PL
W82.00 BOOL  ; STACKING HOOK BACKWARD
W82.01 BOOL  ; STACKING HOOK FORWARD
W82.02 BOOL  ; STACKING LIFTER DOWNWARD
W82.03 BOOL  ; STACKING LIFTER UPWARD
W82.04 BOOL  ; STACKING CONVEYOR
W82.05 BOOL  ; CONVEYOR STOP
W82.06 BOOL  ; STACKING STOPPER DOWNWARD
W82.07 BOOL  ; STACKING STOPPER UPWARD
W82.08 BOOL  ; UNLOADING CONVEYOR 1
W82.10 BOOL  ; UNLOADING ESCAPE UPWARD
W82.11 BOOL  ; UNLOADING ESCAPE DOWNWARD
W82.12 BOOL  ; UNLOADING CONVEYOR 2
W82.14 BOOL  ; UNLOADING STOPPER DOWNWARD
W82.15 BOOL  ; UNLOADING STOPPER UPWARD
W83.00 BOOL  ; STACKING HOOK BACKWARD END
W83.01 BOOL  ; STACKING HOOK FORWARD END
W83.02 BOOL  ; STACKING LIFTER DOWNWARD END
W83.03 BOOL  ; STACKING LIFTER UPWARD END
W83.04 BOOL  ; STACKING CONVEYOR
W83.05 BOOL  ; CONVEYOR STOP
W83.06 BOOL  ; STACKING STOPPER DOWNWARD END
W83.07 BOOL  ; STACKING STOPPER UPWARD END
W83.08 BOOL  ; UNLOADING CONVEYOR 1
W83.10 BOOL  ; UNLOADING ESCAPE UPWARD END
W83.11 BOOL  ; UNLOADING ESCAPE DOWNWARD END
W83.12 BOOL  ; UNLOADING CONVEYOR 2
W83.14 BOOL  ; UNLOADING STOPPER DOWNWARD END
W83.15 BOOL  ; UNLOADING STOPPER UPWARD END
W84.10 BOOL  ; 20ST_1CY START PB
W84.11 BOOL  ; 20ST_1CY RUN PL
W84.12 BOOL  ; 20ST_UNIT HOME POSITION RETURN PB
W84.13 BOOL  ; 20ST_UNIT HOME POSITION PL
W8.00 BOOL  ; Dimension master alignment mode (LM) selection PB
W8.01 BOOL  ; Dimension master alignment mode (S) selection PB
W8.02 BOOL  ; ROBOT MASTER ON
W8.03 BOOL  ; ROBOT FIXED POSITION RETURN
W8.04 BOOL  ; Equipment single operation mode selection PB
W8.05 BOOL  ; BEARING SUPPLY ROBOT FIXID POSITION RETURN
W8.06 BOOL  ; Master work flow mode selection PB
W8.07 BOOL  ; 全作業終了PB
W8.08 BOOL  ; ID RESET START SELECT OF LANE 1
W8.09 BOOL  ; FINISHING OPERATION START
W9.00 BOOL  ; Dimension master matching mode (LM) is being selected
W9.01 BOOL  ; Dimension master matching mode (S) selected PL
W9.02 BOOL  ; ROBOT MASTER ON
W9.03 BOOL  ; ROBOT FIXED POSITION
W9.04 BOOL  ; Equipment unit operation mode selected PL
W9.05 BOOL  ; BEARING FIXID POSITION PL
W9.06 BOOL  ; Master work flow mode selected PL
W9.07 BOOL  ; 全作業終了運転中
W9.08 BOOL  ; ID RESET START SELECT OF LANE 1
W9.09 BOOL  ; FINISHING OPERATION START
B_WorkClampNotUse W303.12 BOOL
BearingInsert_Edit W303.06 BOOL
Bearing_Exchange_Edit W303.11 BOOL
Bearing_Insert_No_Operation W10.11 BOOL
Carrier_Edit W303.01 BOOL  ; Carrier Transfer Edit for BF43
Data_Feed W303.13 BOOL
Fault_Off W303.10 BOOL
Impulse_Edit W303.02 BOOL
LengthMeas_Edit W303.04 BOOL  ; LengthMeas_Edir
Loading_Edit W303.07 BOOL
Master_Check W303.14 BOOL
RB01_DSIN1 3250.00 BOOL  ; Step stop (all tasks)
RB01_DSIN2 3250.01 BOOL  ; <Reserved>
RB01_DSIN3 3250.02 BOOL  ; Instant stop (all tasks)
RB01_DSIN4 3250.03 BOOL  ; Strobe signal
RB01_DSIN5 3250.04 BOOL  ; Interrupt skip
RB01_DSIN6 3250.07 BOOL  ; Command data area odd parity
RB01_DSOUT10 3350.09 BOOL  ; Continue start permission
RB01_DSOUT11 3350.10 BOOL  ; SS mode
RB01_DSOUT12 3350.11 BOOL  ; '-<Reserved>
RB01_DSOUT13 3350.12 BOOL  ; '-<Reserved>
RB01_DSOUT14 3350.13 BOOL  ; '-<Reserved>
RB01_DSOUT15 3350.14 BOOL  ; Command processing complete
RB01_DSOUT16 3350.15 BOOL  ; Status area odd parity
RB01_DSOUT2 3350.01 BOOL  ; During robot operation
RB01_DSOUT3 3350.02 BOOL  ; Robot abnormality
RB01_DSOUT4 3350.03 BOOL  ; Servo on
RB01_DSOUT5 3350.04 BOOL  ; Robot initialization complete
RB01_DSOUT6 3350.05 BOOL  ; Auto mode
RB01_DSOUT7 3350.06 BOOL  ; External mode
RB01_DSOUT8 3350.07 BOOL  ; Battery out warning
RB01_DSOUT9 3350.08 BOOL  ; Robot warning
RB01_DUIN0 3252.07 BOOL
RB01_DUIN1 3252.08 BOOL  ; GRIPPER CLAMP CONFIRM
RB01_DUIN10 3253.01 BOOL
RB01_DUIN100 3258.11 BOOL
RB01_DUIN101 3258.12 BOOL
RB01_DUIN102 3258.13 BOOL
RB01_DUIN103 3258.14 BOOL
RB01_DUIN104 3258.15 BOOL
RB01_DUIN11 3253.02 BOOL
RB01_DUIN12 3253.03 BOOL
RB01_DUIN13 3253.04 BOOL
RB01_DUIN14 3253.05 BOOL
RB01_DUIN15 3253.06 BOOL
RB01_DUIN16 3253.07 BOOL
RB01_DUIN17 3253.08 BOOL
RB01_DUIN18 3253.09 BOOL
RB01_DUIN19 3253.10 BOOL
RB01_DUIN2 3252.09 BOOL  ; GRIPPER UNCLAMP CONFIRM
RB01_DUIN20 3253.11 BOOL
RB01_DUIN21 3253.12 BOOL
RB01_DUIN22 3253.13 BOOL
RB01_DUIN23 3253.14 BOOL
RB01_DUIN24 3253.15 BOOL
RB01_DUIN25 3254.00 BOOL  ; Take Out In Transfer Unit Operation Condition
RB01_DUIN26 3254.01 BOOL  ; Take Out In Transfer Unit No Operation Condition
RB01_DUIN27 3254.02 BOOL  ; Robot Down Operation Good Condition
RB01_DUIN28 3254.03 BOOL  ; Take Out Work Chuck  Operation Complete
RB01_DUIN29 3254.04 BOOL  ; Take Out Operation OK
RB01_DUIN3 3252.10 BOOL  ; LOADING WORKPIECE
RB01_DUIN30 3254.05 BOOL  ; Take Out  Operation NG
RB01_DUIN31 3254.06 BOOL
RB01_DUIN32 3254.07 BOOL
RB01_DUIN33 3254.08 BOOL
RB01_DUIN34 3254.09 BOOL
RB01_DUIN35 3254.10 BOOL
RB01_DUIN36 3254.11 BOOL
RB01_DUIN37 3254.12 BOOL
RB01_DUIN38 3254.13 BOOL
RB01_DUIN39 3254.14 BOOL
RB01_DUIN4 3252.11 BOOL  ; POSITION NUMBER READING START
RB01_DUIN40 3254.15 BOOL
RB01_DUIN41 3255.00 BOOL  ; Take In Work To PalletTizing 1 Operation Condition
RB01_DUIN42 3255.01 BOOL  ; Take In Work To PalletTizing 1  NO Operation Condition
RB01_DUIN43 3255.02 BOOL  ; Robot Down Operation Good Condition
RB01_DUIN44 3255.03 BOOL  ; Take In Work Unchuck Operation Complete
RB01_DUIN45 3255.04 BOOL  ; Take In Work Operation OK
RB01_DUIN46 3255.05 BOOL  ; Take In Work Operation NG
RB01_DUIN47 3255.06 BOOL  ; Removal PalletTizing 1 Clear Request
RB01_DUIN48 3255.07 BOOL  ; Removal Pallet Exchange Recept
RB01_DUIN49 3255.08 BOOL
RB01_DUIN5 3252.12 BOOL
RB01_DUIN50 3255.09 BOOL
RB01_DUIN51 3255.10 BOOL
RB01_DUIN52 3255.11 BOOL
RB01_DUIN53 3255.12 BOOL
RB01_DUIN54 3255.13 BOOL
RB01_DUIN55 3255.14 BOOL
RB01_DUIN56 3255.15 BOOL
RB01_DUIN57 3256.00 BOOL  ; NG Discharge Operation Condition
RB01_DUIN58 3256.01 BOOL  ; NG Discharge NO Operation Condition
RB01_DUIN59 3256.02 BOOL  ; Robot Down Operation Good Condition
RB01_DUIN6 3252.13 BOOL
RB01_DUIN60 3256.03 BOOL  ; NG Discharge Work Unchuck Operation Complete
RB01_DUIN61 3256.04 BOOL  ; NG Discharge Operation OK
RB01_DUIN62 3256.05 BOOL  ; NG Discharge Operation NG
RB01_DUIN63 3256.06 BOOL
RB01_DUIN64 3256.07 BOOL
RB01_DUIN65 3256.08 BOOL
RB01_DUIN66 3256.09 BOOL
RB01_DUIN67 3256.10 BOOL
RB01_DUIN68 3256.11 BOOL
RB01_DUIN69 3256.12 BOOL
RB01_DUIN7 3252.14 BOOL
RB01_DUIN70 3256.13 BOOL
RB01_DUIN71 3256.14 BOOL
RB01_DUIN72 3256.15 BOOL
RB01_DUIN73 3257.00 BOOL  ; LS_Gripper Chuck Confirm
RB01_DUIN74 3257.01 BOOL  ; LS_Gripper UnChuck Confirm
RB01_DUIN75 3257.02 BOOL
RB01_DUIN76 3257.03 BOOL
RB01_DUIN77 3257.04 BOOL
RB01_DUIN78 3257.05 BOOL
RB01_DUIN79 3257.06 BOOL
RB01_DUIN8 3252.15 BOOL
RB01_DUIN80 3257.07 BOOL
RB01_DUIN81 3257.08 BOOL
RB01_DUIN82 3257.09 BOOL
RB01_DUIN83 3257.10 BOOL
RB01_DUIN84 3257.11 BOOL
RB01_DUIN85 3257.12 BOOL
RB01_DUIN86 3257.13 BOOL
RB01_DUIN87 3257.14 BOOL
RB01_DUIN88 3257.15 BOOL
RB01_DUIN89 3258.00 BOOL  ; Take In Work To PalletTizing 2 Operation Condition
RB01_DUIN9 3253.00 BOOL
RB01_DUIN90 3258.01 BOOL  ; Take In Work To PalletTizing 2  NO Operation Condition
RB01_DUIN91 3258.02 BOOL  ; Robot Down Operation Good Condition
RB01_DUIN92 3258.03 BOOL  ; Take In Work Unchuck Operation Complete
RB01_DUIN93 3258.04 BOOL  ; Take In Work Operation OK
RB01_DUIN94 3258.05 BOOL  ; Take In Work Operation NG
RB01_DUIN95 3258.06 BOOL  ; Removal PalletTizing 2 Clear Request
RB01_DUIN96 3258.07 BOOL  ; Removal Pallet Exchange Recept
RB01_DUIN97 3258.08 BOOL
RB01_DUIN98 3258.09 BOOL
RB01_DUIN99 3258.10 BOOL
RB01_DUOUT1 3352.00 BOOL  ; Robot fixed position
RB01_DUOUT10 3352.09 BOOL  ; Reservation
RB01_DUOUT100 3358.03 BOOL  ; Removal PalletTizing 2 Clear Completed
RB01_DUOUT101 3358.04 BOOL  ; Removal magazine replacement command
RB01_DUOUT102 3358.05 BOOL
RB01_DUOUT103 3358.06 BOOL
RB01_DUOUT104 3358.07 BOOL
RB01_DUOUT105 3358.08 BOOL
RB01_DUOUT106 3358.09 BOOL
RB01_DUOUT107 3358.10 BOOL
RB01_DUOUT108 3358.11 BOOL
RB01_DUOUT109 3358.12 BOOL
RB01_DUOUT11 3352.10 BOOL  ; Reservation
RB01_DUOUT110 3358.13 BOOL
RB01_DUOUT111 3358.14 BOOL
RB01_DUOUT112 3358.15 BOOL
RB01_DUOUT12 3352.11 BOOL  ; Reservation
RB01_DUOUT13 3352.12 BOOL  ; Reservation
RB01_DUOUT14 3352.13 BOOL  ; Signal reading timing in area
RB01_DUOUT15 3352.14 BOOL  ; In robot area
RB01_DUOUT16 3352.15 BOOL  ; Reservation
RB01_DUOUT2 3352.01 BOOL  ; Transfer data received
RB01_DUOUT3 3352.02 BOOL  ; Motor On
RB01_DUOUT33 3354.00 BOOL  ; Take Out In Transfer Unit No Operation Condition
RB01_DUOUT34 3354.01 BOOL  ; Removal work chuck operation completed
RB01_DUOUT35 3354.02 BOOL  ; Take Out operation completed
RB01_DUOUT36 3354.03 BOOL
RB01_DUOUT37 3354.04 BOOL
RB01_DUOUT38 3354.05 BOOL
RB01_DUOUT39 3354.06 BOOL
RB01_DUOUT4 3352.03 BOOL  ; Program End
RB01_DUOUT40 3354.07 BOOL
RB01_DUOUT41 3354.08 BOOL
RB01_DUOUT42 3354.09 BOOL
RB01_DUOUT43 3354.10 BOOL
RB01_DUOUT44 3354.11 BOOL
RB01_DUOUT45 3354.12 BOOL
RB01_DUOUT46 3354.13 BOOL
RB01_DUOUT47 3354.14 BOOL
RB01_DUOUT48 3354.15 BOOL
RB01_DUOUT49 3355.00 BOOL  ; Take In Work To Pallet1Tizing 1 No Operation Condition
RB01_DUOUT5 3352.04 BOOL  ; Robot Operation Fault
RB01_DUOUT50 3355.01 BOOL  ; Take In  work unchuck op. completed
RB01_DUOUT51 3355.02 BOOL  ; Take In Work To PalletTizing 1  Operation Complete
RB01_DUOUT52 3355.03 BOOL  ; Removal PalletTizing 1 Clear Completed
RB01_DUOUT53 3355.04 BOOL  ; Removal magazine replacement command
RB01_DUOUT54 3355.05 BOOL
RB01_DUOUT55 3355.06 BOOL
RB01_DUOUT56 3355.07 BOOL
RB01_DUOUT57 3355.08 BOOL
RB01_DUOUT58 3355.09 BOOL
RB01_DUOUT59 3355.10 BOOL
RB01_DUOUT6 3352.05 BOOL  ; Parts chuck in progress
RB01_DUOUT60 3355.11 BOOL
RB01_DUOUT61 3355.12 BOOL
RB01_DUOUT62 3355.13 BOOL
RB01_DUOUT63 3355.14 BOOL
RB01_DUOUT64 3355.15 BOOL
RB01_DUOUT65 3356.00 BOOL  ; NG Discharge No Operation Condition
RB01_DUOUT66 3356.01 BOOL  ; NG Discharge work unchuck operation completed
RB01_DUOUT67 3356.02 BOOL  ; NG Discharge Operation Complete
RB01_DUOUT68 3356.03 BOOL
RB01_DUOUT69 3356.04 BOOL
RB01_DUOUT7 3352.06 BOOL  ; Sensor check NG
RB01_DUOUT70 3356.05 BOOL
RB01_DUOUT71 3356.06 BOOL
RB01_DUOUT72 3356.07 BOOL
RB01_DUOUT73 3356.08 BOOL
RB01_DUOUT74 3356.09 BOOL
RB01_DUOUT75 3356.10 BOOL
RB01_DUOUT76 3356.11 BOOL
RB01_DUOUT77 3356.12 BOOL
RB01_DUOUT78 3356.13 BOOL
RB01_DUOUT79 3356.14 BOOL
RB01_DUOUT8 3352.07 BOOL  ; Hand exchange NG
RB01_DUOUT80 3356.15 BOOL
RB01_DUOUT81 3357.00 BOOL  ; Sol_Gripper Chuck
RB01_DUOUT82 3357.01 BOOL  ; Sol_Gripper UnChuck
RB01_DUOUT83 3357.02 BOOL
RB01_DUOUT84 3357.03 BOOL
RB01_DUOUT85 3357.04 BOOL
RB01_DUOUT86 3357.05 BOOL
RB01_DUOUT87 3357.06 BOOL
RB01_DUOUT88 3357.07 BOOL
RB01_DUOUT89 3357.08 BOOL
RB01_DUOUT9 3352.08 BOOL  ; Visual judgment NG
RB01_DUOUT90 3357.09 BOOL
RB01_DUOUT91 3357.10 BOOL
RB01_DUOUT92 3357.11 BOOL
RB01_DUOUT93 3357.12 BOOL
RB01_DUOUT94 3357.13 BOOL
RB01_DUOUT95 3357.14 BOOL
RB01_DUOUT96 3357.15 BOOL
RB01_DUOUT97 3358.00 BOOL  ; Take In Work To Pallet1Tizing 2 No Operation Condition
RB01_DUOUT98 3358.01 BOOL  ; Take In  work unchuck op. completed
RB01_DUOUT99 3358.02 BOOL  ; Take In Work To PalletTizing 2  Operation Complete
RB1_edit W303.00 BOOL  ; Robot Change Program (RC5=>RC8)
Resistance_Counting_ProbeNG W10.14 BOOL
Resistance_Edit W303.03 BOOL
Whitout_Part W303.09 BOOL

## Program MainProgram (cyclic task 0)

### Section Adjustment

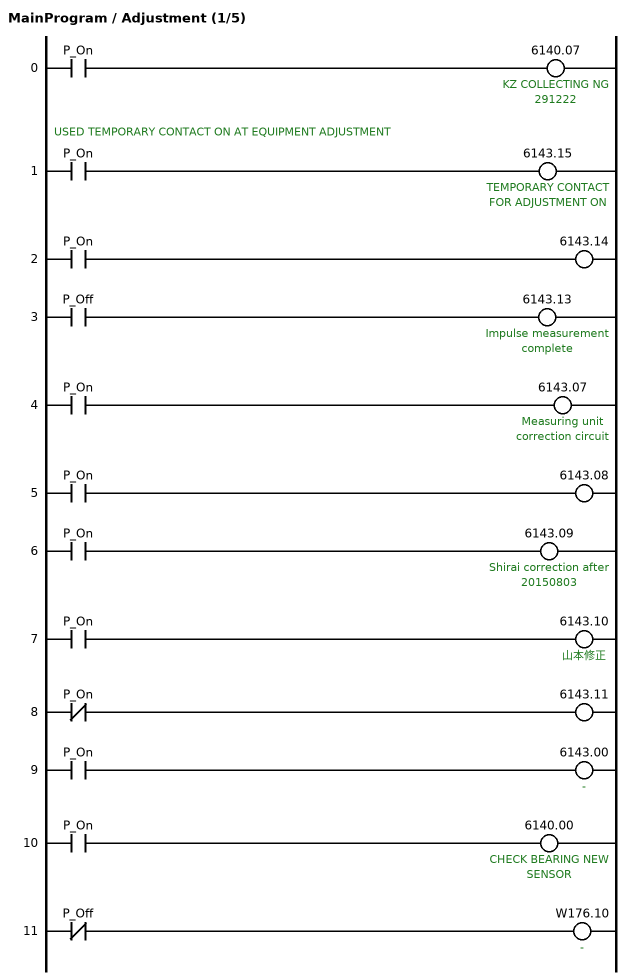
; rung 0
LD P_On
OUT 6140.07  ; KZ COLLECTING NG 291222
; rung 1: USED TEMPORARY CONTACT ON AT EQUIPMENT ADJUSTMENT
LD P_On
OUT 6143.15  ; TEMPORARY CONTACT FOR ADJUSTMENT ON
; rung 2
LD P_On
OUT 6143.14
; rung 3
LD P_Off
OUT 6143.13  ; Impulse measurement complete
; rung 4
LD P_On
OUT 6143.07  ; Measuring unit correction circuit
; rung 5
LD P_On
OUT 6143.08
; rung 6
LD P_On
OUT 6143.09  ; Shirai correction after 20150803
; rung 7
LD P_On
OUT 6143.10  ; 山本修正
; rung 8
LDNOT P_On
OUT 6143.11
; rung 9
LD P_On
OUT 6143.00  ; -
; rung 10
LD P_On
OUT 6140.00  ; CHECK BEARING NEW SENSOR
; rung 11
LDNOT P_Off
OUT W176.10  ; -

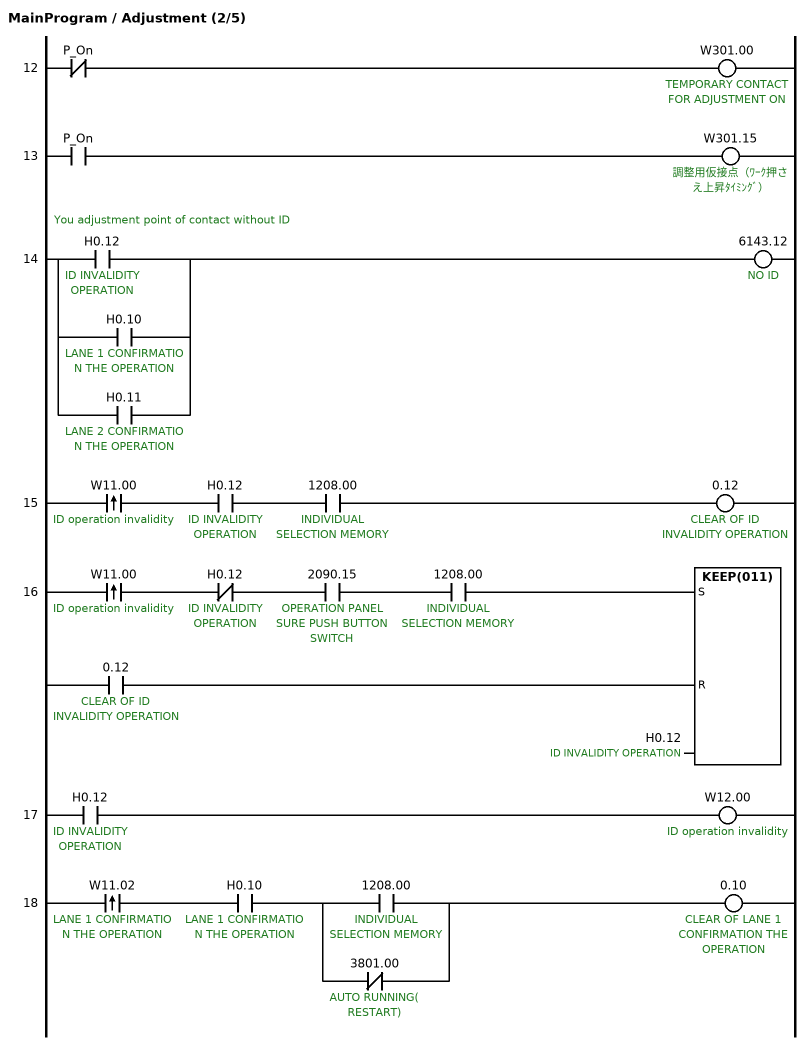
; rung 12
LDNOT P_On
OUT W301.00  ; TEMPORARY CONTACT FOR ADJUSTMENT ON
; rung 13
LD P_On
OUT W301.15  ; 調整用仮接点（ﾜｰｸ押さえ上昇ﾀｲﾐﾝｸﾞ）
; rung 14: You adjustment point of contact without ID
LD H0.12  ; ID INVALIDITY OPERATION
OR H0.10  ; LANE 1 CONFIRMATION THE OPERATION
OR H0.11  ; LANE 2 CONFIRMATION THE OPERATION
OUT 6143.12  ; NO ID
; rung 15
@LD W11.00  ; ID operation invalidity
AND H0.12  ; ID INVALIDITY OPERATION
AND 1208.00  ; INDIVIDUAL SELECTION MEMORY
OUT 0.12  ; CLEAR OF ID INVALIDITY OPERATION
; rung 16
@LD W11.00  ; ID operation invalidity
ANDNOT H0.12  ; ID INVALIDITY OPERATION
AND 2090.15  ; OPERATION PANEL SURE PUSH BUTTON SWITCH
AND 1208.00  ; INDIVIDUAL SELECTION MEMORY
LD 0.12  ; CLEAR OF ID INVALIDITY OPERATION
KEEP(011) H0.12  ; ID INVALIDITY OPERATION
; rung 17
LD H0.12  ; ID INVALIDITY OPERATION
OUT W12.00  ; ID operation invalidity
; rung 18
@LD W11.02  ; LANE 1 CONFIRMATION THE OPERATION
AND H0.10  ; LANE 1 CONFIRMATION THE OPERATION
LD 1208.00  ; INDIVIDUAL SELECTION MEMORY
ORNOT 3801.00  ; AUTO RUNNING(RESTART)
ANDLD
OUT 0.10  ; CLEAR OF LANE 1 CONFIRMATION THE OPERATION

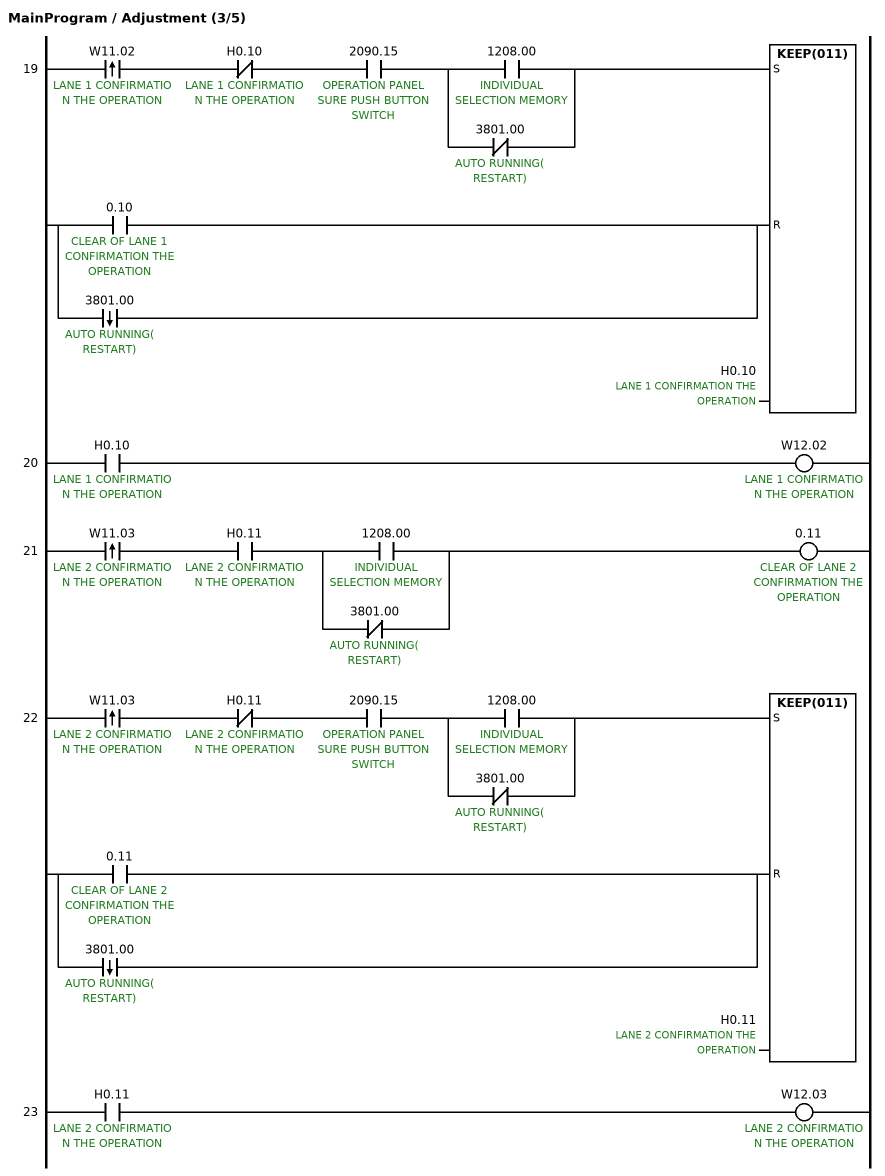
; rung 19
@LD W11.02  ; LANE 1 CONFIRMATION THE OPERATION
ANDNOT H0.10  ; LANE 1 CONFIRMATION THE OPERATION
AND 2090.15  ; OPERATION PANEL SURE PUSH BUTTON SWITCH
LD 1208.00  ; INDIVIDUAL SELECTION MEMORY
ORNOT 3801.00  ; AUTO RUNNING(RESTART)
ANDLD
LD 0.10  ; CLEAR OF LANE 1 CONFIRMATION THE OPERATION
%OR 3801.00  ; AUTO RUNNING(RESTART)
KEEP(011) H0.10  ; LANE 1 CONFIRMATION THE OPERATION
; rung 20
LD H0.10  ; LANE 1 CONFIRMATION THE OPERATION
OUT W12.02  ; LANE 1 CONFIRMATION THE OPERATION
; rung 21
@LD W11.03  ; LANE 2 CONFIRMATION THE OPERATION
AND H0.11  ; LANE 2 CONFIRMATION THE OPERATION
LD 1208.00  ; INDIVIDUAL SELECTION MEMORY
ORNOT 3801.00  ; AUTO RUNNING(RESTART)
ANDLD
OUT 0.11  ; CLEAR OF LANE 2 CONFIRMATION THE OPERATION
; rung 22
@LD W11.03  ; LANE 2 CONFIRMATION THE OPERATION
ANDNOT H0.11  ; LANE 2 CONFIRMATION THE OPERATION
AND 2090.15  ; OPERATION PANEL SURE PUSH BUTTON SWITCH
LD 1208.00  ; INDIVIDUAL SELECTION MEMORY
ORNOT 3801.00  ; AUTO RUNNING(RESTART)
ANDLD
LD 0.11  ; CLEAR OF LANE 2 CONFIRMATION THE OPERATION
%OR 3801.00  ; AUTO RUNNING(RESTART)
KEEP(011) H0.11  ; LANE 2 CONFIRMATION THE OPERATION
; rung 23
LD H0.11  ; LANE 2 CONFIRMATION THE OPERATION
OUT W12.03  ; LANE 2 CONFIRMATION THE OPERATION

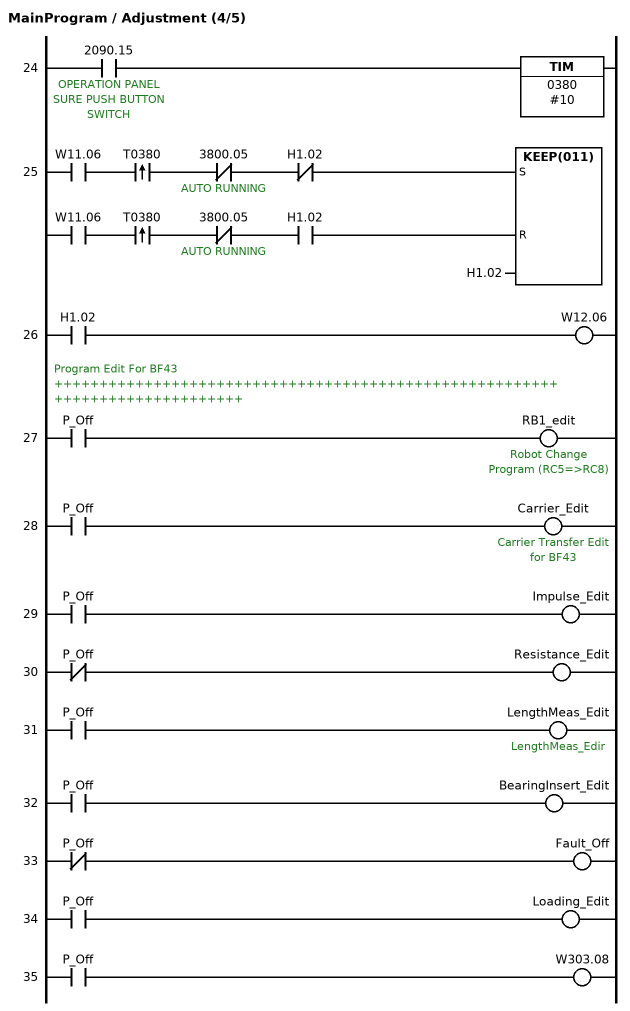
; rung 24
LD 2090.15  ; OPERATION PANEL SURE PUSH BUTTON SWITCH
TIM 0380 #10
; rung 25
LD W11.06
@AND T0380
ANDNOT 3800.05  ; AUTO RUNNING
ANDNOT H1.02
LD W11.06
@AND T0380
ANDNOT 3800.05  ; AUTO RUNNING
AND H1.02
KEEP(011) H1.02
; rung 26
LD H1.02
OUT W12.06
; rung 27: Program Edit For BF43 / +++++++++++++++++++++++++++++++++++++++++++++++++++++++++++++++++++++++++++++
LD P_Off
OUT RB1_edit  ; Robot Change Program (RC5=>RC8)
; rung 28
LD P_Off
OUT Carrier_Edit  ; Carrier Transfer Edit for BF43
; rung 29
LD P_Off
OUT Impulse_Edit
; rung 30
LDNOT P_Off
OUT Resistance_Edit
; rung 31
LD P_Off
OUT LengthMeas_Edit  ; LengthMeas_Edir
; rung 32
LD P_Off
OUT BearingInsert_Edit
; rung 33
LDNOT P_Off
OUT Fault_Off
; rung 34
LD P_Off
OUT Loading_Edit
; rung 35
LD P_Off
OUT W303.08

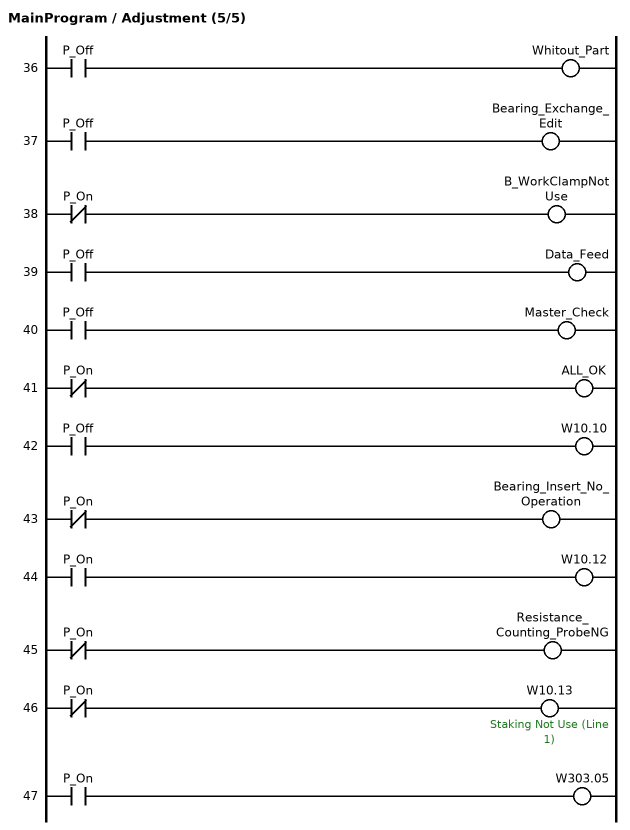
; rung 36
LD P_Off
OUT Whitout_Part
; rung 37
LD P_Off
OUT Bearing_Exchange_Edit
; rung 38
LDNOT P_On
OUT B_WorkClampNotUse
; rung 39
LD P_Off
OUT Data_Feed
; rung 40
LD P_Off
OUT Master_Check
; rung 41
LDNOT P_On
OUT ALL_OK
; rung 42
LD P_Off
OUT W10.10
; rung 43
LDNOT P_On
OUT Bearing_Insert_No_Operation
; rung 44
LD P_On
OUT W10.12
; rung 45
LDNOT P_On
OUT Resistance_Counting_ProbeNG
; rung 46
LDNOT P_On
OUT W10.13  ; Staking Not Use (Line 1)
; rung 47
LD P_On
OUT W303.05

### Section Data_for_resistance_and_impulse_measurement

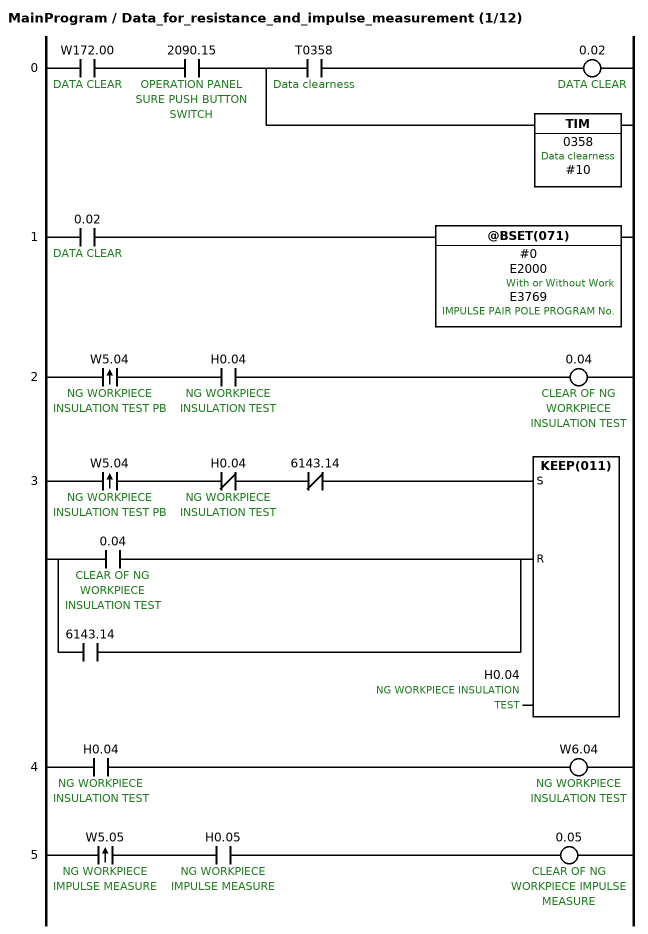
; rung 0
LD W172.00  ; DATA CLEAR
AND 2090.15  ; OPERATION PANEL SURE PUSH BUTTON SWITCH
OUT TR0
AND T0358  ; Data clearness
OUT 0.02  ; DATA CLEAR
LD TR0
TIM 0358 #10  ; Data clearness
; rung 1
LD 0.02  ; DATA CLEAR
@BSET(071) #0 E2000 E3769  ; With or Without Work, IMPULSE PAIR POLE PROGRAM No.
; rung 2
@LD W5.04  ; NG WORKPIECE INSULATION TEST PB
AND H0.04  ; NG WORKPIECE INSULATION TEST
OUT 0.04  ; CLEAR OF NG WORKPIECE INSULATION TEST
; rung 3
@LD W5.04  ; NG WORKPIECE INSULATION TEST PB
ANDNOT H0.04  ; NG WORKPIECE INSULATION TEST
ANDNOT 6143.14
LD 0.04  ; CLEAR OF NG WORKPIECE INSULATION TEST
OR 6143.14
KEEP(011) H0.04  ; NG WORKPIECE INSULATION TEST
; rung 4
LD H0.04  ; NG WORKPIECE INSULATION TEST
OUT W6.04  ; NG WORKPIECE INSULATION TEST
; rung 5
@LD W5.05  ; NG WORKPIECE IMPULSE MEASURE
AND H0.05  ; NG WORKPIECE IMPULSE MEASURE
OUT 0.05  ; CLEAR OF NG WORKPIECE IMPULSE MEASURE

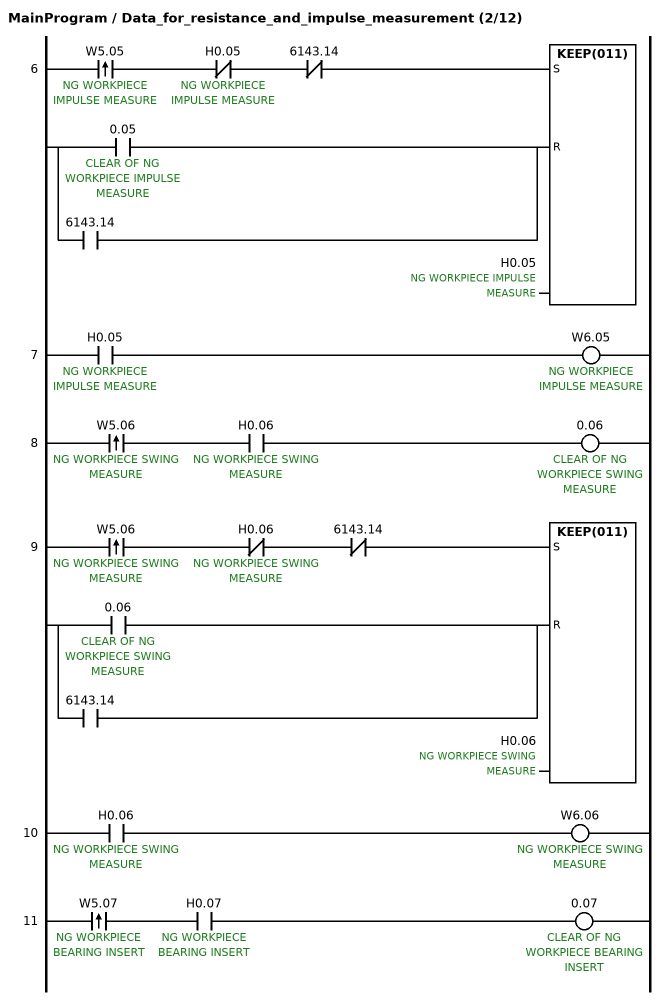
; rung 6
@LD W5.05  ; NG WORKPIECE IMPULSE MEASURE
ANDNOT H0.05  ; NG WORKPIECE IMPULSE MEASURE
ANDNOT 6143.14
LD 0.05  ; CLEAR OF NG WORKPIECE IMPULSE MEASURE
OR 6143.14
KEEP(011) H0.05  ; NG WORKPIECE IMPULSE MEASURE
; rung 7
LD H0.05  ; NG WORKPIECE IMPULSE MEASURE
OUT W6.05  ; NG WORKPIECE IMPULSE MEASURE
; rung 8
@LD W5.06  ; NG WORKPIECE SWING MEASURE
AND H0.06  ; NG WORKPIECE SWING MEASURE
OUT 0.06  ; CLEAR OF NG WORKPIECE SWING MEASURE
; rung 9
@LD W5.06  ; NG WORKPIECE SWING MEASURE
ANDNOT H0.06  ; NG WORKPIECE SWING MEASURE
ANDNOT 6143.14
LD 0.06  ; CLEAR OF NG WORKPIECE SWING MEASURE
OR 6143.14
KEEP(011) H0.06  ; NG WORKPIECE SWING MEASURE
; rung 10
LD H0.06  ; NG WORKPIECE SWING MEASURE
OUT W6.06  ; NG WORKPIECE SWING MEASURE
; rung 11
@LD W5.07  ; NG WORKPIECE BEARING INSERT
AND H0.07  ; NG WORKPIECE BEARING INSERT
OUT 0.07  ; CLEAR OF NG WORKPIECE BEARING INSERT

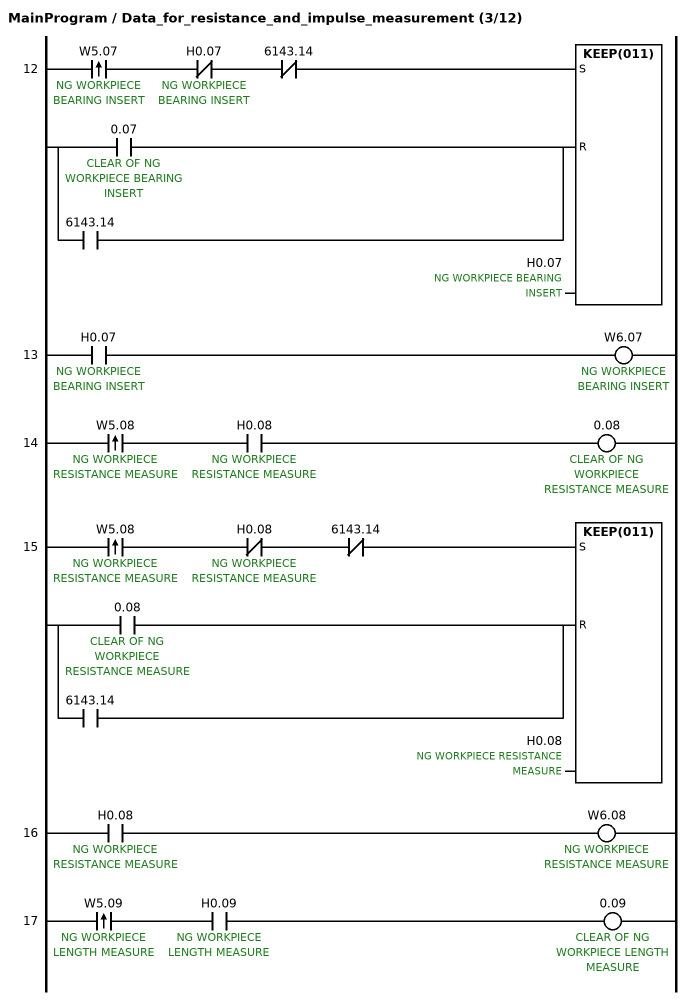
; rung 12
@LD W5.07  ; NG WORKPIECE BEARING INSERT
ANDNOT H0.07  ; NG WORKPIECE BEARING INSERT
ANDNOT 6143.14
LD 0.07  ; CLEAR OF NG WORKPIECE BEARING INSERT
OR 6143.14
KEEP(011) H0.07  ; NG WORKPIECE BEARING INSERT
; rung 13
LD H0.07  ; NG WORKPIECE BEARING INSERT
OUT W6.07  ; NG WORKPIECE BEARING INSERT
; rung 14
@LD W5.08  ; NG WORKPIECE RESISTANCE MEASURE
AND H0.08  ; NG WORKPIECE RESISTANCE MEASURE
OUT 0.08  ; CLEAR OF NG WORKPIECE RESISTANCE MEASURE
; rung 15
@LD W5.08  ; NG WORKPIECE RESISTANCE MEASURE
ANDNOT H0.08  ; NG WORKPIECE RESISTANCE MEASURE
ANDNOT 6143.14
LD 0.08  ; CLEAR OF NG WORKPIECE RESISTANCE MEASURE
OR 6143.14
KEEP(011) H0.08  ; NG WORKPIECE RESISTANCE MEASURE
; rung 16
LD H0.08  ; NG WORKPIECE RESISTANCE MEASURE
OUT W6.08  ; NG WORKPIECE RESISTANCE MEASURE
; rung 17
@LD W5.09  ; NG WORKPIECE LENGTH MEASURE
AND H0.09  ; NG WORKPIECE LENGTH MEASURE
OUT 0.09  ; CLEAR OF NG WORKPIECE LENGTH MEASURE

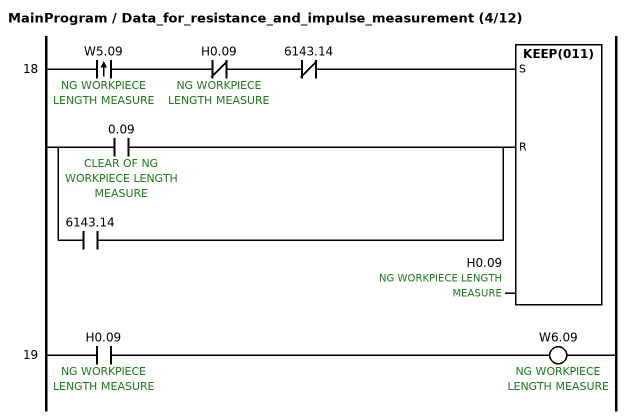
; rung 18
@LD W5.09  ; NG WORKPIECE LENGTH MEASURE
ANDNOT H0.09  ; NG WORKPIECE LENGTH MEASURE
ANDNOT 6143.14
LD 0.09  ; CLEAR OF NG WORKPIECE LENGTH MEASURE
OR 6143.14
KEEP(011) H0.09  ; NG WORKPIECE LENGTH MEASURE
; rung 19
LD H0.09  ; NG WORKPIECE LENGTH MEASURE
OUT W6.09  ; NG WORKPIECE LENGTH MEASURE

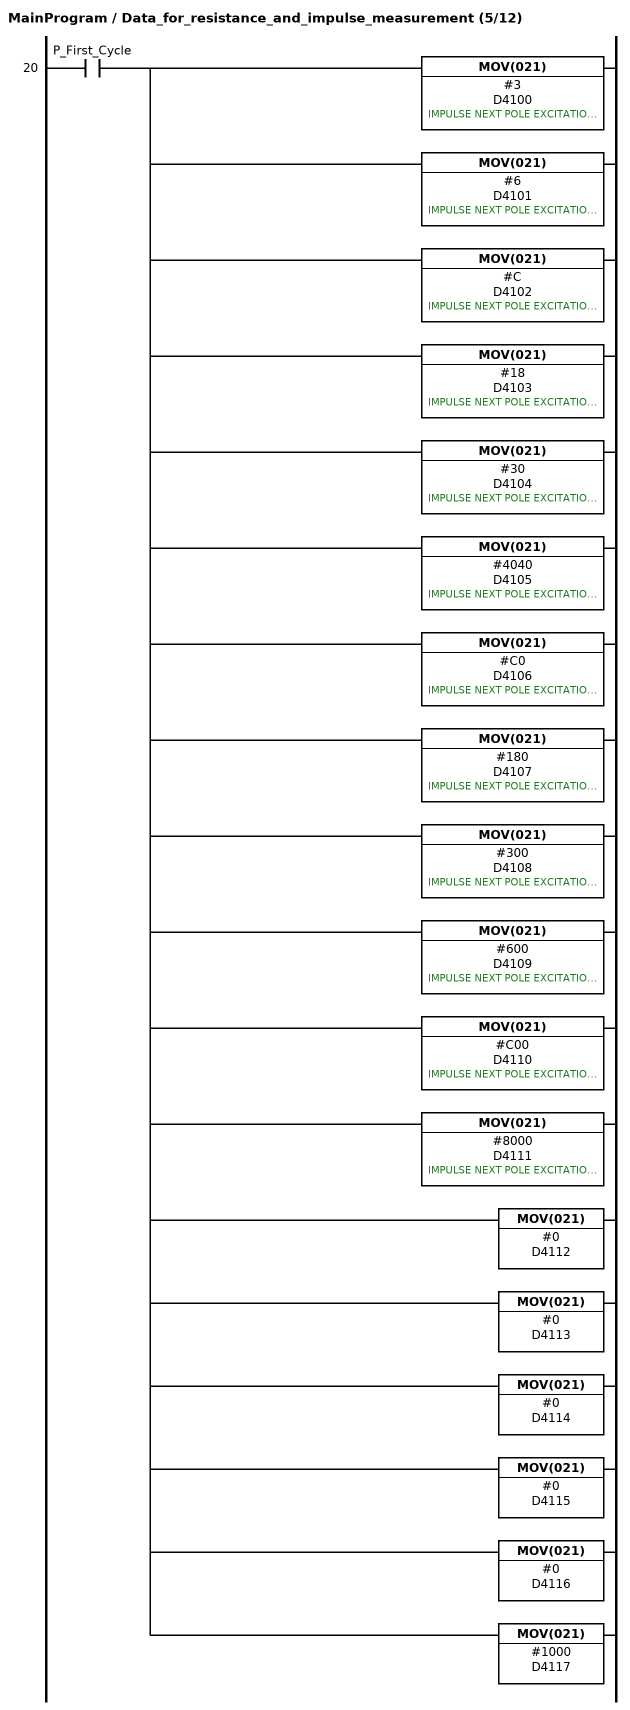
; rung 20
LD P_First_Cycle
MOV(021) #3 D4100  ; IMPULSE NEXT POLE EXCITATION PATTERN 1-2
MOV(021) #6 D4101  ; IMPULSE NEXT POLE EXCITATION PATTERN 2-3
MOV(021) #C D4102  ; IMPULSE NEXT POLE EXCITATION PATTERN 3-4
MOV(021) #18 D4103  ; IMPULSE NEXT POLE EXCITATION PATTERN 4-5
MOV(021) #30 D4104  ; IMPULSE NEXT POLE EXCITATION PATTERN 5-6
MOV(021) #4040 D4105  ; IMPULSE NEXT POLE EXCITATION PATTERN 6-7
MOV(021) #C0 D4106  ; IMPULSE NEXT POLE EXCITATION PATTERN 7-8
MOV(021) #180 D4107  ; IMPULSE NEXT POLE EXCITATION PATTERN 8-9
MOV(021) #300 D4108  ; IMPULSE NEXT POLE EXCITATION PATTERN 9-10
MOV(021) #600 D4109  ; IMPULSE NEXT POLE EXCITATION PATTERN 10-11
MOV(021) #C00 D4110  ; IMPULSE NEXT POLE EXCITATION PATTERN 10-12
MOV(021) #8000 D4111  ; IMPULSE NEXT POLE EXCITATION PATTERN 12-1
MOV(021) #0 D4112
MOV(021) #0 D4113
MOV(021) #0 D4114
MOV(021) #0 D4115
MOV(021) #0 D4116
MOV(021) #1000 D4117

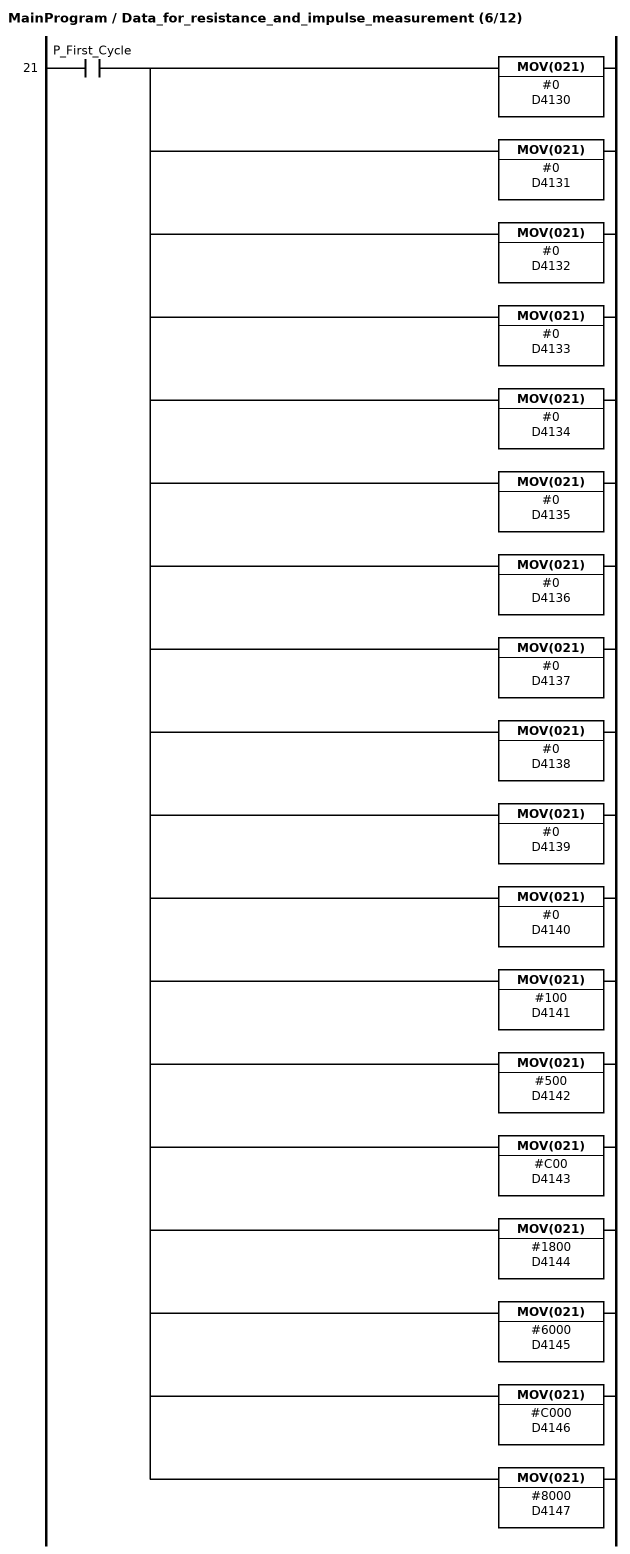
; rung 21
LD P_First_Cycle
MOV(021) #0 D4130
MOV(021) #0 D4131
MOV(021) #0 D4132
MOV(021) #0 D4133
MOV(021) #0 D4134
MOV(021) #0 D4135
MOV(021) #0 D4136
MOV(021) #0 D4137
MOV(021) #0 D4138
MOV(021) #0 D4139
MOV(021) #0 D4140
MOV(021) #100 D4141
MOV(021) #500 D4142
MOV(021) #C00 D4143
MOV(021) #1800 D4144
MOV(021) #6000 D4145
MOV(021) #C000 D4146
MOV(021) #8000 D4147

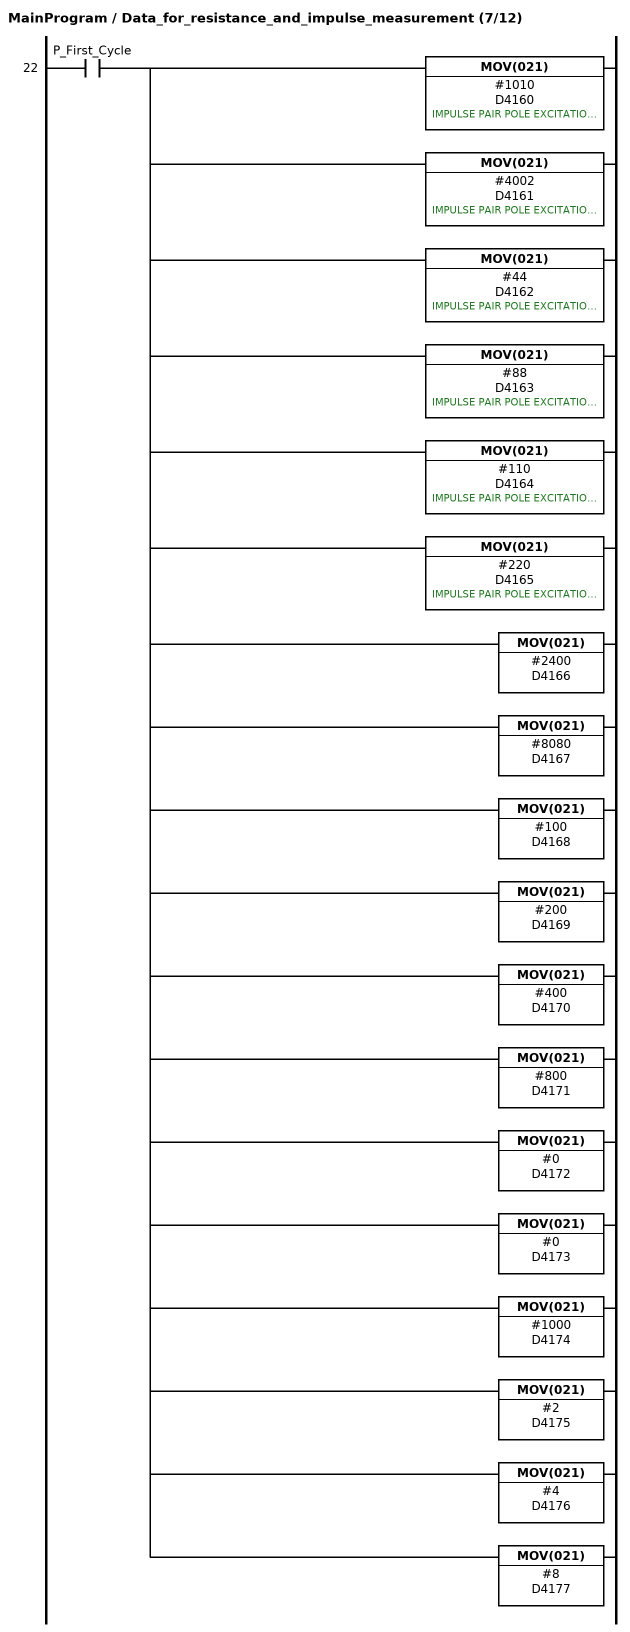
; rung 22
LD P_First_Cycle
MOV(021) #1010 D4160  ; IMPULSE PAIR POLE EXCITATION PATTERN 1-7  // IMPULSE PAIR POLE EXCITATION PATTERN 1-5
MOV(021) #4002 D4161  ; IMPULSE PAIR POLE EXCITATION PATTERN 2-8  // IMPULSE PAIR POLE EXCITATION PATTERN 2-6
MOV(021) #44 D4162  ; IMPULSE PAIR POLE EXCITATION PATTERN 3-9  // IMPULSE PAIR POLE EXCITATION PATTERN 3-7
MOV(021) #88 D4163  ; IMPULSE PAIR POLE EXCITATION PATTERN 4-10  // IMPULSE PAIR POLE EXCITATION PATTERN 4-8
MOV(021) #110 D4164  ; IMPULSE PAIR POLE EXCITATION PATTERN 5-11  // IMPULSE PAIR POLE EXCITATION PATTERN 4-9
MOV(021) #220 D4165  ; IMPULSE PAIR POLE EXCITATION PATTERN 6-12  // IMPULSE PAIR POLE EXCITATION PATTERN 6-10
MOV(021) #2400 D4166  // IMPULSE PAIR POLE EXCITATION PATTERN 7-11
MOV(021) #8080 D4167  // IMPULSE PAIR POLE EXCITATION PATTERN 8-12
MOV(021) #100 D4168  // IMPULSE PAIR POLE EXCITATION PATTERN 9-13
MOV(021) #200 D4169  // IMPULSE PAIR POLE EXCITATION PATTERN 10-14
MOV(021) #400 D4170  // IMPULSE PAIR POLE EXCITATION PATTERN 11-15
MOV(021) #800 D4171  // IMPULSE PAIR POLE EXCITATION PATTERN 12-16
MOV(021) #0 D4172  // IMPULSE PAIR POLE EXCITATION PATTERN 13-17
MOV(021) #0 D4173  // IMPULSE PAIR POLE EXCITATION PATTERN 14-18
MOV(021) #1000 D4174  // IMPULSE PAIR POLE EXCITATION PATTERN 15-1
MOV(021) #2 D4175  // IMPULSE PAIR POLE EXCITATION PATTERN 16-2
MOV(021) #4 D4176  // IMPULSE PAIR POLE EXCITATION PATTERN 3-17
MOV(021) #8 D4177  // IMPULSE PAIR POLE EXCITATION PATTERN 18-4

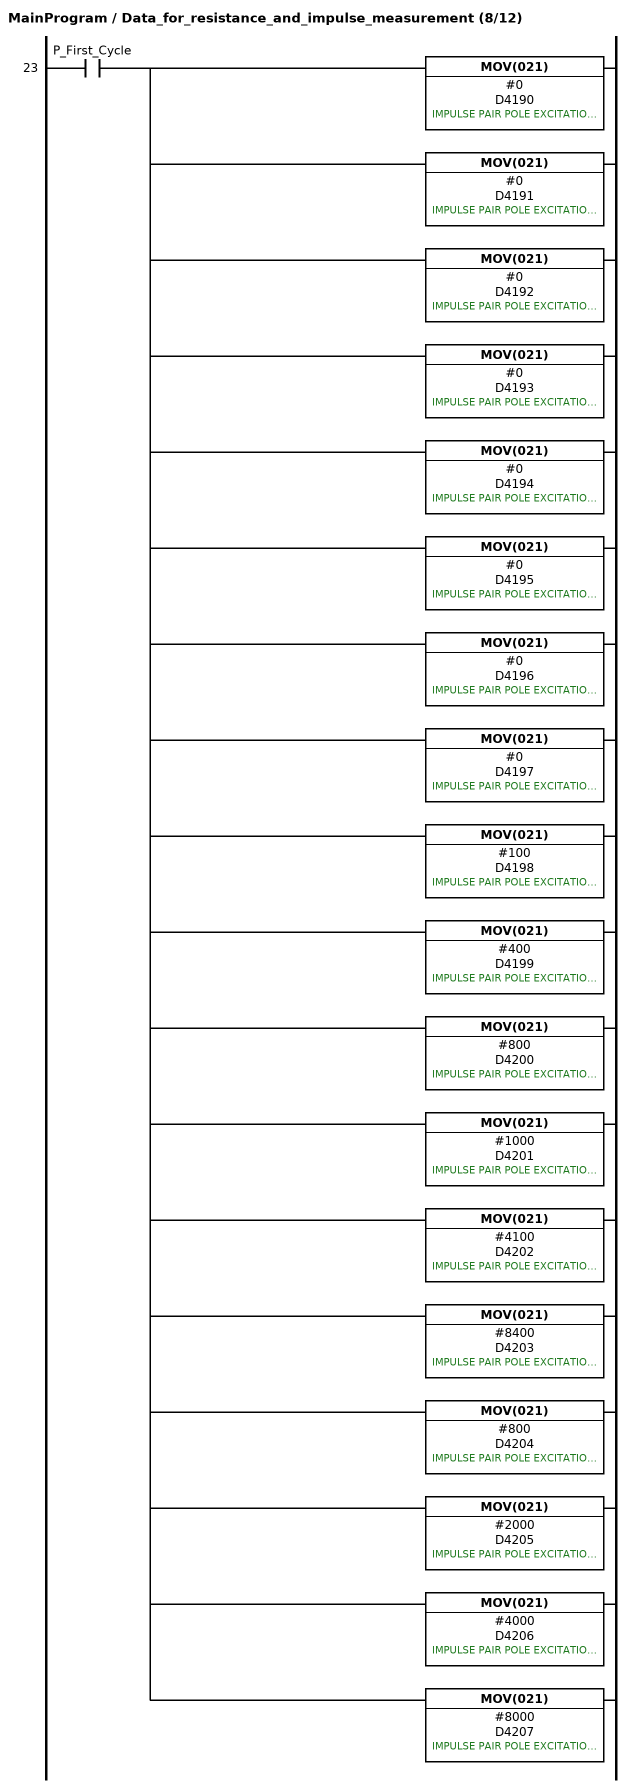
; rung 23
LD P_First_Cycle
MOV(021) #0 D4190  ; IMPULSE PAIR POLE EXCITATION PATTERN 1-5
MOV(021) #0 D4191  ; IMPULSE PAIR POLE EXCITATION PATTERN 2-6
MOV(021) #0 D4192  ; IMPULSE PAIR POLE EXCITATION PATTERN 3-7
MOV(021) #0 D4193  ; IMPULSE PAIR POLE EXCITATION PATTERN 4-8
MOV(021) #0 D4194  ; IMPULSE PAIR POLE EXCITATION PATTERN 5-9
MOV(021) #0 D4195  ; IMPULSE PAIR POLE EXCITATION PATTERN 6-10
MOV(021) #0 D4196  ; IMPULSE PAIR POLE EXCITATION PATTERN 7-11
MOV(021) #0 D4197  ; IMPULSE PAIR POLE EXCITATION PATTERN 8-12
MOV(021) #100 D4198  ; IMPULSE PAIR POLE EXCITATION PATTERN 9-13
MOV(021) #400 D4199  ; IMPULSE PAIR POLE EXCITATION PATTERN 10-14
MOV(021) #800 D4200  ; IMPULSE PAIR POLE EXCITATION PATTERN 11-15
MOV(021) #1000 D4201  ; IMPULSE PAIR POLE EXCITATION PATTERN 12-16
MOV(021) #4100 D4202  ; IMPULSE PAIR POLE EXCITATION PATTERN 13-17
MOV(021) #8400 D4203  ; IMPULSE PAIR POLE EXCITATION PATTERN 14-18
MOV(021) #800 D4204  ; IMPULSE PAIR POLE EXCITATION PATTERN 15-1
MOV(021) #2000 D4205  ; IMPULSE PAIR POLE EXCITATION PATTERN 16-2
MOV(021) #4000 D4206  ; IMPULSE PAIR POLE EXCITATION PATTERN 17-3
MOV(021) #8000 D4207  ; IMPULSE PAIR POLE EXCITATION PATTERN 18-1

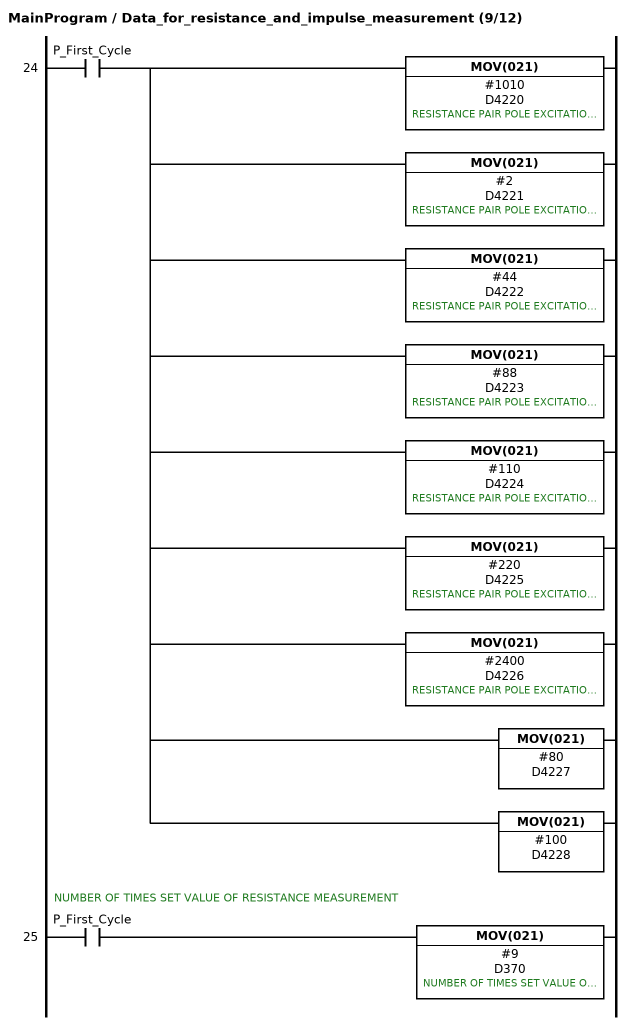
; rung 24
LD P_First_Cycle
MOV(021) #1010 D4220  ; RESISTANCE PAIR POLE EXCITATION PATTERN 1-7  // RESISTANCE PAIR POLE EXCITATION PATTERN 1-5
MOV(021) #2 D4221  ; RESISTANCE PAIR POLE EXCITATION PATTERN 2-8  // RESISTANCE PAIR POLE EXCITATION PATTERN 2-6
MOV(021) #44 D4222  ; RESISTANCE PAIR POLE EXCITATION PATTERN 3-9  // RESISTANCE PAIR POLE EXCITATION PATTERN 3-7
MOV(021) #88 D4223  ; RESISTANCE PAIR POLE EXCITATION PATTERN 4-10  // RESISTANCE PAIR POLE EXCITATION PATTERN 4-8
MOV(021) #110 D4224  ; RESISTANCE PAIR POLE EXCITATION PATTERN 5-11  // RESISTANCE PAIR POLE EXCITATION PATTERN 5-9
MOV(021) #220 D4225  ; RESISTANCE PAIR POLE EXCITATION PATTERN 6-12  // RESISTANCE PAIR POLE EXCITATION PATTERN 6-10
MOV(021) #2400 D4226  ; RESISTANCE PAIR POLE EXCITATION PATTERN 7-11  // RESISTANCE PAIR POLE EXCITATION PATTERN 7-11
MOV(021) #80 D4227  // RESISTANCE PAIR POLE EXCITATION PATTERN 8-12
MOV(021) #100 D4228  // RESISTANCE PAIR POLE EXCITATION PATTERN 9-13
; rung 25: NUMBER OF TIMES SET VALUE OF RESISTANCE MEASUREMENT
LD P_First_Cycle
MOV(021) #9 D370  ; NUMBER OF TIMES SET VALUE OF RESISTANCE MEASUREMENT  // 80 Degree

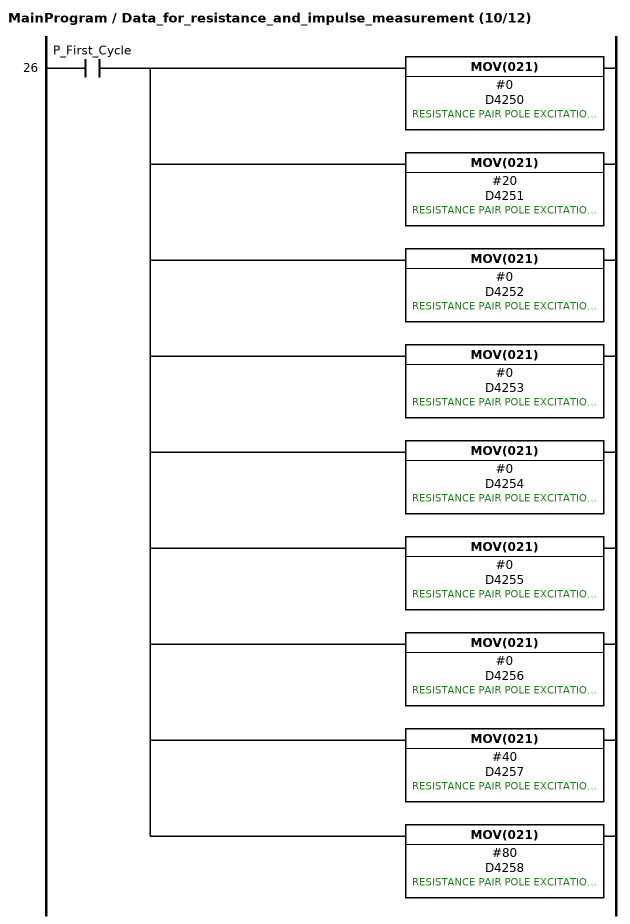
; rung 26
LD P_First_Cycle
MOV(021) #0 D4250  ; RESISTANCE PAIR POLE EXCITATION PATTERN 1-5
MOV(021) #20 D4251  ; RESISTANCE PAIR POLE EXCITATION PATTERN 2-6
MOV(021) #0 D4252  ; RESISTANCE PAIR POLE EXCITATION PATTERN 3-7
MOV(021) #0 D4253  ; RESISTANCE PAIR POLE EXCITATION PATTERN 4-8
MOV(021) #0 D4254  ; RESISTANCE PAIR POLE EXCITATION PATTERN 5-9
MOV(021) #0 D4255  ; RESISTANCE PAIR POLE EXCITATION PATTERN 6-10
MOV(021) #0 D4256  ; RESISTANCE PAIR POLE EXCITATION PATTERN 7-11
MOV(021) #40 D4257  ; RESISTANCE PAIR POLE EXCITATION PATTERN 8-12
MOV(021) #80 D4258  ; RESISTANCE PAIR POLE EXCITATION PATTERN 9-13

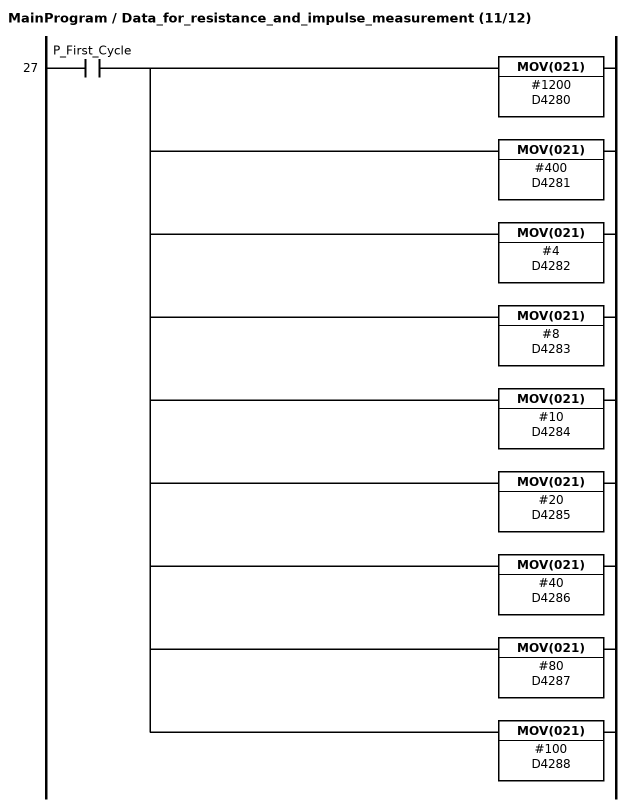
; rung 27
LD P_First_Cycle
MOV(021) #1200 D4280
MOV(021) #400 D4281
MOV(021) #4 D4282
MOV(021) #8 D4283
MOV(021) #10 D4284
MOV(021) #20 D4285
MOV(021) #40 D4286
MOV(021) #80 D4287
MOV(021) #100 D4288

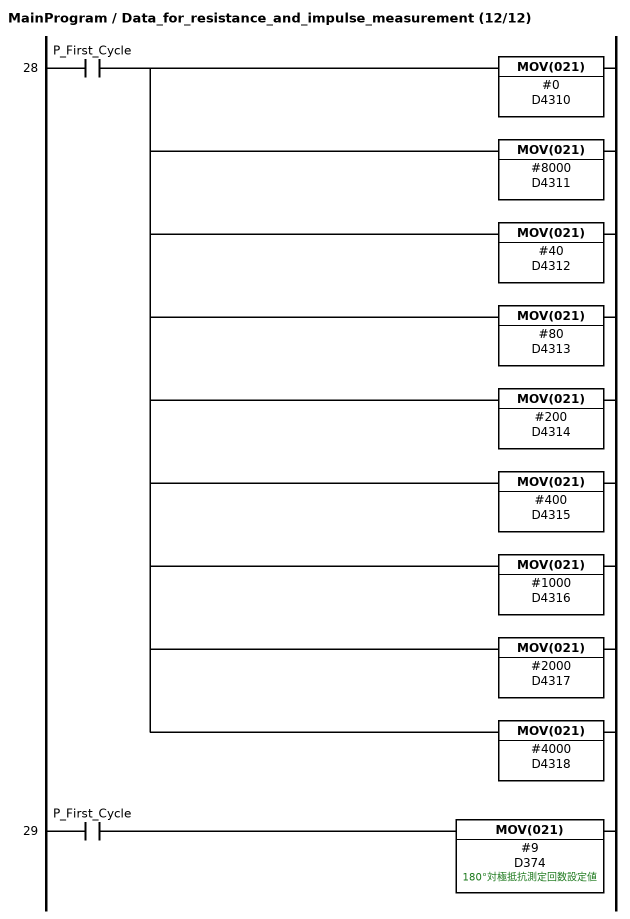
; rung 28
LD P_First_Cycle
MOV(021) #0 D4310
MOV(021) #8000 D4311
MOV(021) #40 D4312
MOV(021) #80 D4313
MOV(021) #200 D4314
MOV(021) #400 D4315
MOV(021) #1000 D4316
MOV(021) #2000 D4317
MOV(021) #4000 D4318
; rung 29
LD P_First_Cycle
MOV(021) #9 D374  ; 180°対極抵抗測定回数設定値  // 180 Degree

### Section MASTER_ON_CIRCUIT_BOARD_PL

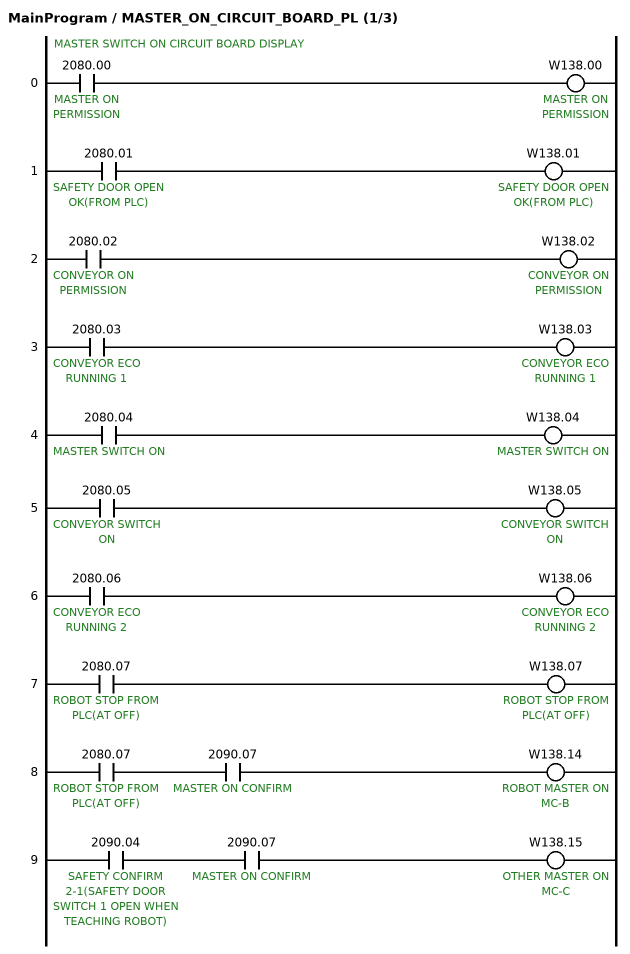
; rung 0: MASTER SWITCH ON CIRCUIT BOARD DISPLAY
LD 2080.00  ; MASTER ON PERMISSION
OUT W138.00  ; MASTER ON PERMISSION
; rung 1
LD 2080.01  ; SAFETY DOOR OPEN OK(FROM PLC)
OUT W138.01  ; SAFETY DOOR OPEN OK(FROM PLC)
; rung 2
LD 2080.02  ; CONVEYOR ON PERMISSION
OUT W138.02  ; CONVEYOR ON PERMISSION
; rung 3
LD 2080.03  ; CONVEYOR ECO RUNNING 1
OUT W138.03  ; CONVEYOR ECO RUNNING 1
; rung 4
LD 2080.04  ; MASTER SWITCH ON
OUT W138.04  ; MASTER SWITCH ON
; rung 5
LD 2080.05  ; CONVEYOR SWITCH ON
OUT W138.05  ; CONVEYOR SWITCH ON
; rung 6
LD 2080.06  ; CONVEYOR ECO RUNNING 2
OUT W138.06  ; CONVEYOR ECO RUNNING 2
; rung 7
LD 2080.07  ; ROBOT STOP FROM PLC(AT OFF)
OUT W138.07  ; ROBOT STOP FROM PLC(AT OFF)
; rung 8
LD 2080.07  ; ROBOT STOP FROM PLC(AT OFF)
AND 2090.07  ; MASTER ON CONFIRM
OUT W138.14  ; ROBOT MASTER ON MC-B
; rung 9
LD 2090.04  ; SAFETY CONFIRM 2-1(SAFETY DOOR SWITCH 1 OPEN WHEN TEACHING ROBOT)
AND 2090.07  ; MASTER ON CONFIRM
OUT W138.15  ; OTHER MASTER ON MC-C

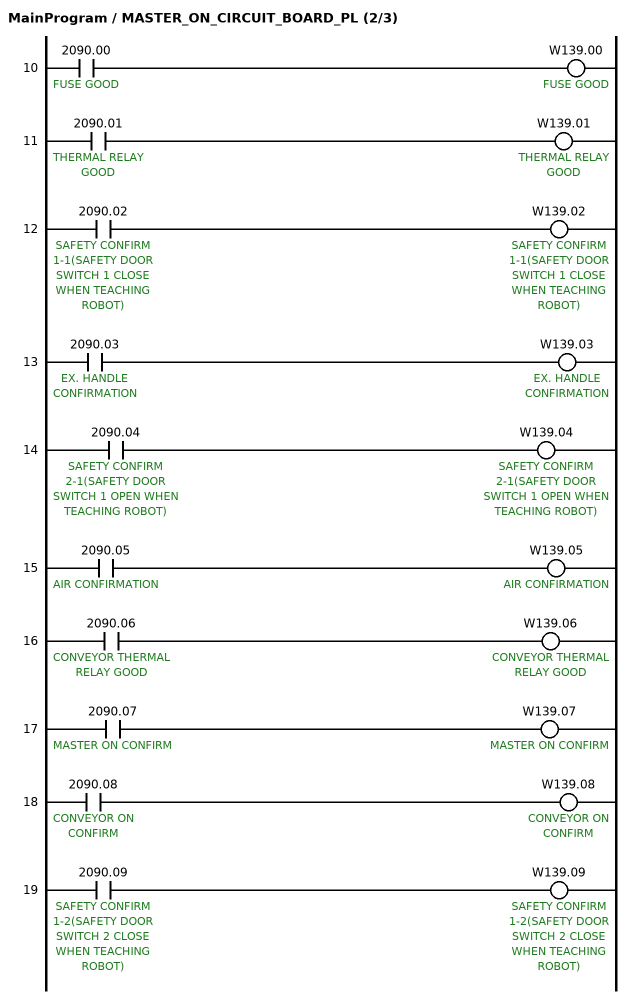
; rung 10
LD 2090.00  ; FUSE GOOD
OUT W139.00  ; FUSE GOOD
; rung 11
LD 2090.01  ; THERMAL RELAY GOOD
OUT W139.01  ; THERMAL RELAY GOOD
; rung 12
LD 2090.02  ; SAFETY CONFIRM 1-1(SAFETY DOOR SWITCH 1 CLOSE WHEN TEACHING ROBOT)
OUT W139.02  ; SAFETY CONFIRM 1-1(SAFETY DOOR SWITCH 1 CLOSE WHEN TEACHING ROBOT)
; rung 13
LD 2090.03  ; EX. HANDLE CONFIRMATION
OUT W139.03  ; EX. HANDLE CONFIRMATION
; rung 14
LD 2090.04  ; SAFETY CONFIRM 2-1(SAFETY DOOR SWITCH 1 OPEN WHEN TEACHING ROBOT)
OUT W139.04  ; SAFETY CONFIRM 2-1(SAFETY DOOR SWITCH 1 OPEN WHEN TEACHING ROBOT)
; rung 15
LD 2090.05  ; AIR CONFIRMATION
OUT W139.05  ; AIR CONFIRMATION
; rung 16
LD 2090.06  ; CONVEYOR THERMAL RELAY GOOD
OUT W139.06  ; CONVEYOR THERMAL RELAY GOOD
; rung 17
LD 2090.07  ; MASTER ON CONFIRM
OUT W139.07  ; MASTER ON CONFIRM
; rung 18
LD 2090.08  ; CONVEYOR ON CONFIRM
OUT W139.08  ; CONVEYOR ON CONFIRM
; rung 19
LD 2090.09  ; SAFETY CONFIRM 1-2(SAFETY DOOR SWITCH 2 CLOSE WHEN TEACHING ROBOT)
OUT W139.09  ; SAFETY CONFIRM 1-2(SAFETY DOOR SWITCH 2 CLOSE WHEN TEACHING ROBOT)

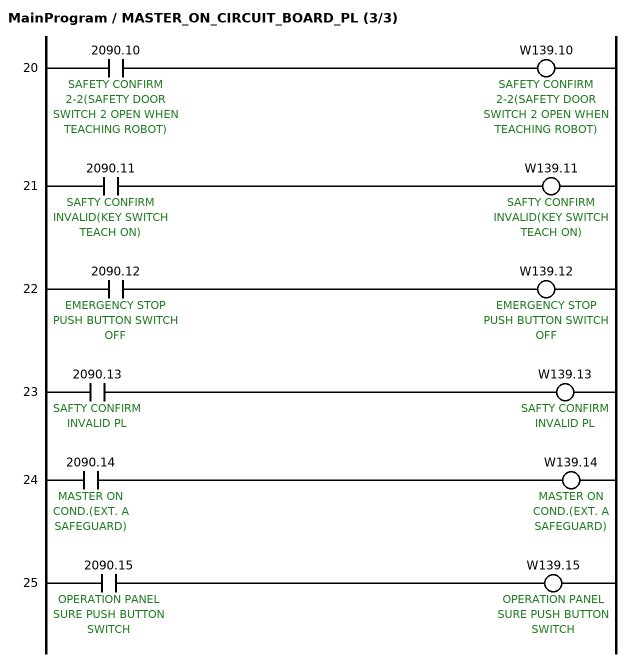
; rung 20
LD 2090.10  ; SAFETY CONFIRM 2-2(SAFETY DOOR SWITCH 2 OPEN WHEN TEACHING ROBOT)
OUT W139.10  ; SAFETY CONFIRM 2-2(SAFETY DOOR SWITCH 2 OPEN WHEN TEACHING ROBOT)
; rung 21
LD 2090.11  ; SAFTY CONFIRM INVALID(KEY SWITCH TEACH ON)
OUT W139.11  ; SAFTY CONFIRM INVALID(KEY SWITCH TEACH ON)
; rung 22
LD 2090.12  ; EMERGENCY STOP PUSH BUTTON SWITCH OFF
OUT W139.12  ; EMERGENCY STOP PUSH BUTTON SWITCH OFF
; rung 23
LD 2090.13  ; SAFTY CONFIRM INVALID PL
OUT W139.13  ; SAFTY CONFIRM INVALID PL
; rung 24
LD 2090.14  ; MASTER ON COND.(EXT. A SAFEGUARD)
OUT W139.14  ; MASTER ON COND.(EXT. A SAFEGUARD)
; rung 25
LD 2090.15  ; OPERATION PANEL SURE PUSH BUTTON SWITCH
OUT W139.15  ; OPERATION PANEL SURE PUSH BUTTON SWITCH

### Section SURE_PB

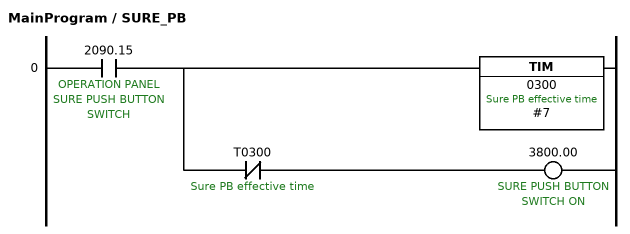
; rung 0
LD 2090.15  ; OPERATION PANEL SURE PUSH BUTTON SWITCH
TIM 0300 #7  ; Sure PB effective time
ANDNOT T0300  ; Sure PB effective time
OUT 3800.00  ; SURE PUSH BUTTON SWITCH ON

### Section Controller_Link_SETUP

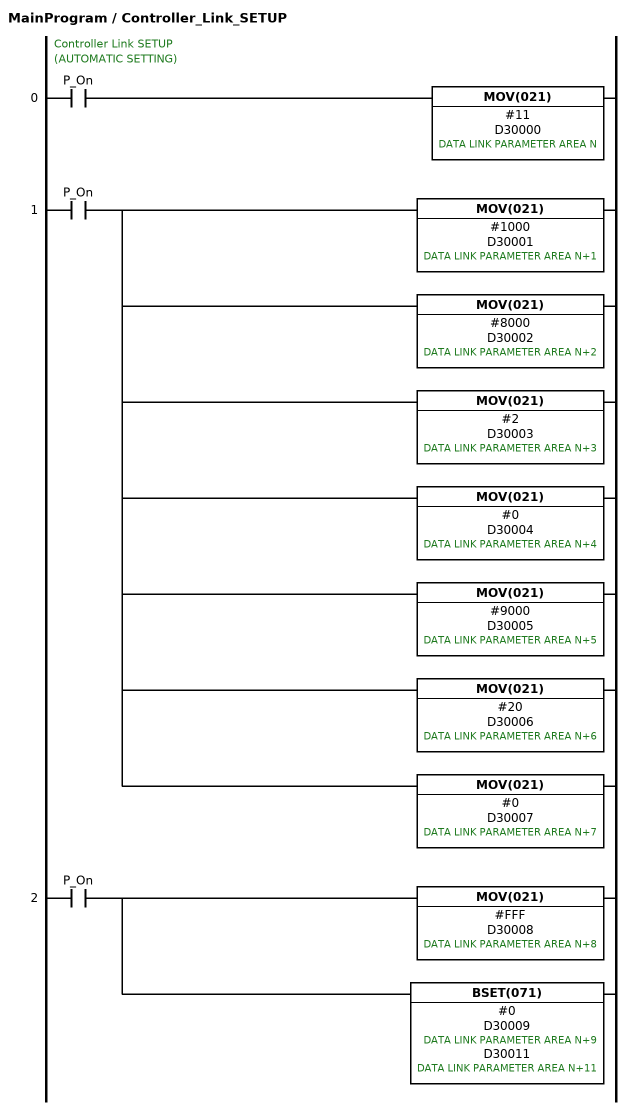
; rung 0: Controller Link SETUP / (AUTOMATIC SETTING)
LD P_On
MOV(021) #11 D30000  ; DATA LINK PARAMETER AREA N  // Setting data links / N:D30000+(100*Controller Link Unit number):F
; rung 1
LD P_On
MOV(021) #1000 D30001  ; DATA LINK PARAMETER AREA N+1  // Area 1 data link start word (BCD)
MOV(021) #8000 D30002  ; DATA LINK PARAMETER AREA N+2  // Area 1 type
MOV(021) #2 D30003  ; DATA LINK PARAMETER AREA N+3  // Number of send words per node of area 1 (BCD)
MOV(021) #0 D30004  ; DATA LINK PARAMETER AREA N+4  // Rightmost 4 digits of data link start word of area 2 (DM area)(BCD)
MOV(021) #9000 D30005  ; DATA LINK PARAMETER AREA N+5  // Area 2 type ; Leftmost digit of data link start word of area 2 (BCD)
MOV(021) #20 D30006  ; DATA LINK PARAMETER AREA N+6  // Number of send words per node of area 2 (BCD)
MOV(021) #0 D30007  ; DATA LINK PARAMETER AREA N+7  // First data link status word (BCD)
; rung 2
LD P_On
MOV(021) #FFF D30008  ; DATA LINK PARAMETER AREA N+8  // Nodes to participate in the data links / The numbers indicate node numbers. / The value assigned indicates whether the node is to perticipate in the data links. / Perticipate: 1     Not perticipate: 0
BSET(071) #0 D30009 D30011  ; DATA LINK PARAMETER AREA N+9, DATA LINK PARAMETER AREA N+11

### Section ID001

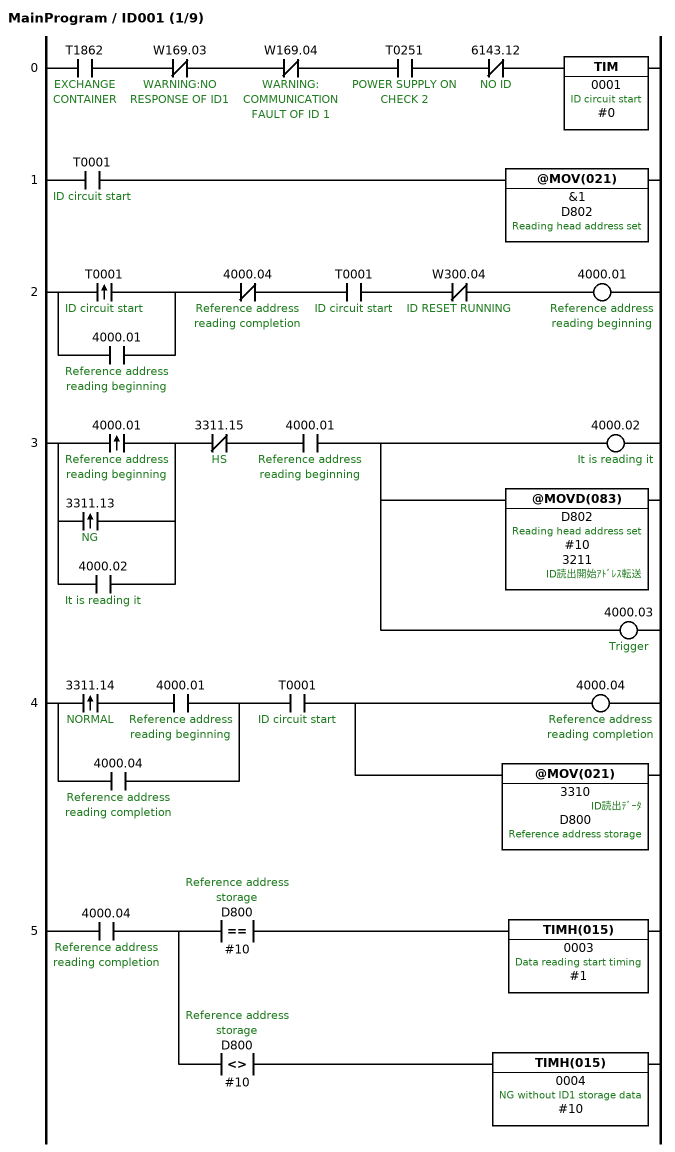
; rung 0
LD T1862  ; EXCHANGE CONTAINER
ANDNOT W169.03  ; WARNING:NO RESPONSE OF ID1
ANDNOT W169.04  ; WARNING:COMMUNICATION FAULT OF ID 1
AND T0251  ; POWER SUPPLY ON CHECK 2
ANDNOT 6143.12  ; NO ID
TIM 0001 #0  ; ID circuit start
; rung 1
LD T0001  ; ID circuit start
@MOV(021) &1 D802  ; Reading head address set
; rung 2
@LD T0001  ; ID circuit start
OR 4000.01  ; Reference address reading beginning
ANDNOT 4000.04  ; Reference address reading completion
AND T0001  ; ID circuit start
ANDNOT W300.04  ; ID RESET RUNNING
OUT 4000.01  ; Reference address reading beginning
; rung 3
@LD 4000.01  ; Reference address reading beginning
@OR 3311.13  ; NG
OR 4000.02  ; It is reading it
ANDNOT 3311.15  ; HS
AND 4000.01  ; Reference address reading beginning
OUT 4000.02  ; It is reading it
@MOVD(083) D802 #10 3211  ; Reading head address set, ID読出開始ｱﾄﾞﾚｽ転送
OUT 4000.03  ; Trigger
; rung 4
@LD 3311.14  ; NORMAL
AND 4000.01  ; Reference address reading beginning
OR 4000.04  ; Reference address reading completion
AND T0001  ; ID circuit start
OUT 4000.04  ; Reference address reading completion
@MOV(021) 3310 D800  ; ID読出ﾃﾞｰﾀ, Reference address storage
; rung 5
LD 4000.04  ; Reference address reading completion
OUT TR0
AND=(300) D800 #10  ; Reference address storage
TIMH(015) 0003 #1  ; Data reading start timing
LD TR0
AND<>(305) D800 #10  ; Reference address storage
TIMH(015) 0004 #10  ; NG without ID1 storage data

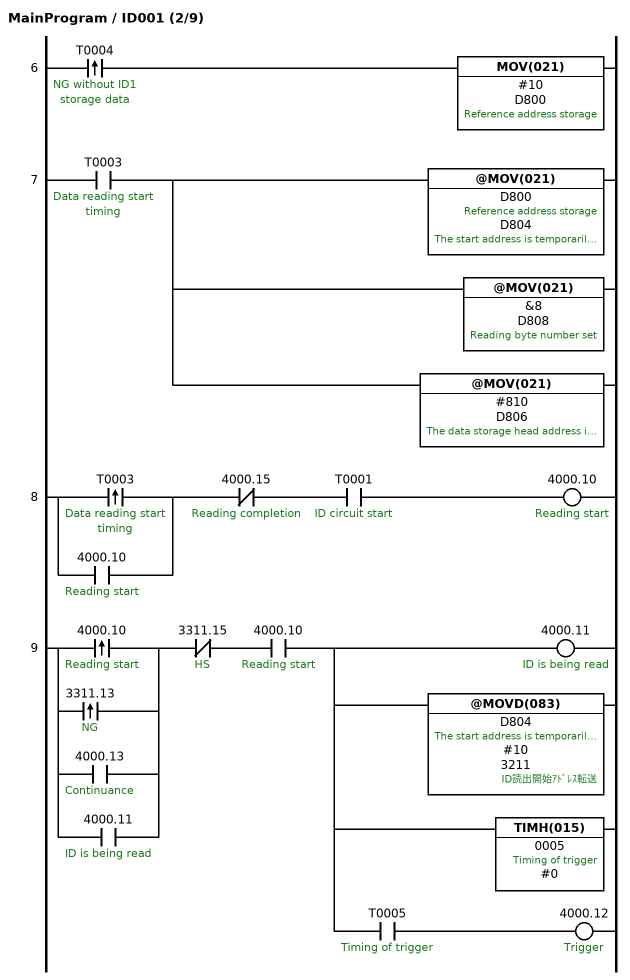
; rung 6
@LD T0004  ; NG without ID1 storage data
MOV(021) #10 D800  ; Reference address storage
; rung 7
LD T0003  ; Data reading start timing
@MOV(021) D800 D804  ; Reference address storage, The start address is temporarily memorized
@MOV(021) &8 D808  ; Reading byte number set
@MOV(021) #810 D806  ; The data storage head address is memorized
; rung 8
@LD T0003  ; Data reading start timing
OR 4000.10  ; Reading start
ANDNOT 4000.15  ; Reading completion
AND T0001  ; ID circuit start
OUT 4000.10  ; Reading start
; rung 9
@LD 4000.10  ; Reading start
@OR 3311.13  ; NG
OR 4000.13  ; Continuance
OR 4000.11  ; ID is being read
ANDNOT 3311.15  ; HS
AND 4000.10  ; Reading start
OUT 4000.11  ; ID is being read
@MOVD(083) D804 #10 3211  ; The start address is temporarily memorized, ID読出開始ｱﾄﾞﾚｽ転送
TIMH(015) 0005 #0  ; Timing of trigger
AND T0005  ; Timing of trigger
OUT 4000.12  ; Trigger

